// ---- GVLs/kitting deca/axis/AxisHMI_Ex.TcVIS
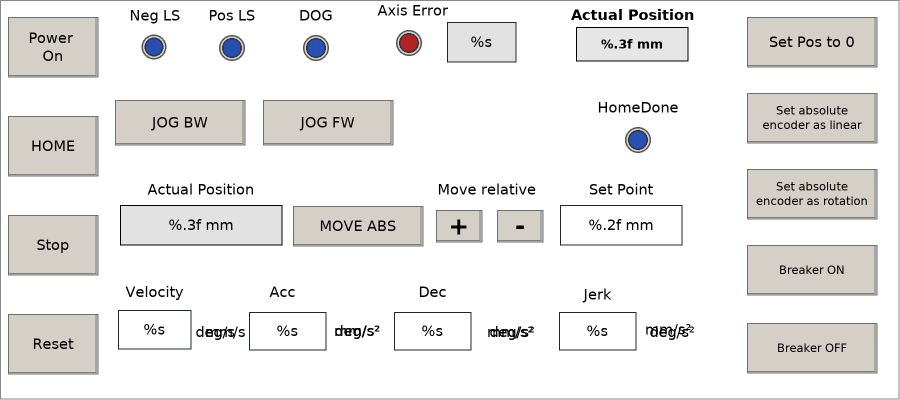
VISUALIZATION AxisHMI_Ex  // 900x400
VAR_IN_OUT
	stAxisHMI	: ST_MotionAxis_MC	;
	mcAxis		: FB_MotionAxis_MC;
	//sAxisName	: STRING			;// Axis Name
	//iAxisID		: INT			;// Axis Id
	xError		: BOOL				;// Axis error flag
END_VAR
    Button (115,100 130x45), "JOG BW", colour toggle: stAxisHMI.mcJog.JogBackwards
        OnMouseDown: execute { stAxisHMI.mcJog.JogBackwards := TRUE; }
        OnMouseUp: execute { stAxisHMI.mcJog.JogBackwards := FALSE; }
    Button (263,100 130x45), "JOG FW", colour toggle: stAxisHMI.mcJog.JogForward
        OnMouseDown: execute { stAxisHMI.mcJog.JogForward := TRUE; }
        OnMouseUp: execute { stAxisHMI.mcJog.JogForward := FALSE; }
    Rectangle (120,205 162x40), "%.3f mm", text variable: stAxisHMI.rActualPosHMI
        OnMouseClick: write the text variable via Default
    Label (141,177 120x25), "Actual Position"
    Button (8,17 90x60), "Power On", colour toggle: stAxisHMI.mcPower.Enable, pressed state: stAxisHMI.mcPower.Enable
        OnMouseClick: toggle stAxisHMI.mcPower.Enable
    Button (8,215 90x60), "Stop", colour toggle: stAxisHMI.mcStop.Execute, invisible if: NOT stAxisHMI.bStopButtonShow
        OnMouseDown: execute { stAxisHMI.mcStop.Execute := TRUE; }
        OnMouseUp: execute { stAxisHMI.mcStop.Execute := FALSE; }
    Button (8,314 90x60), "Reset", colour toggle: stAxisHMI.mcReset.Execute
        OnMouseDown: execute { stAxisHMI.mcReset.Execute := TRUE; }
        OnMouseUp: execute { stAxisHMI.mcReset.Execute := FALSE; }
    Label (111,277 87x30), "Velocity"
    Rectangle (118,310 73x39), "%s", text variable: stAxisHMI.rVeloPers
        OnMouseClick: write the text variable via Default, min 1, max stAxisHMI.rMaxVelocity
    Label (230,277 105x30), "Acc"
    Rectangle (249,312 77x38), "%s", text variable: stAxisHMI.rAcceleration
        OnMouseClick: write stAxisHMI.rAccPers via Default, min 1, max stAxisHMI.rMaxAcceleration
    Lamp1 (139,33 30x28), variable: stAxisHMI.bNegSen, invisible if: NOT stAxisHMI.bNegSensorShow, style: Lamp-Lamp1-Blue
    Label (364,-2 102x25), "Axis Error"
    Rectangle (447,22 69x40), "%s", text variable: stAxisHMI.mcReadStatus.ErrorID
    Lamp1 (394,28 30x30), variable: xError, style: Lamp-Lamp1-Red
    Lamp1 (217,33 30x30), variable: stAxisHMI.bPosSen, invisible if: NOT stAxisHMI.bPosSensorShow, style: Lamp-Lamp1-Blue
    Label (188,3 88x25), "Pos LS", invisible if: NOT stAxisHMI.bPosSensorShow
    Label (111,3 88x25), "Neg LS", invisible if: NOT stAxisHMI.bNegSensorShow
    Rectangle (560,205 122x40), "%.2f mm", text variable: stAxisHMI.rDistance
        OnMouseClick: write the text variable via Default, min 0, max stAxisHMI.rMaxDistance
    Button (293,206 130x40), "MOVE ABS", colour toggle: stAxisHMI.mcMoveAbsolute.Busy, pressed state: stAxisHMI.mcMoveAbsolute.Busy
        OnMouseDown: execute { stAxisHMI.bMoveAbsHMI := TRUE; }
        OnMouseUp: execute { stAxisHMI.bMoveAbsHMI := FALSE; }
    Label (561,177 120x25), "Set Point"
    Button (436,210 46x32), "+", colour toggle: stAxisHMI.mcMoveRelative.Busy, pressed state: stAxisHMI.mcMoveRelative.Busy
        OnMouseDown: execute { stAxisHMI.rPosition := stAxisHMI.rDistance; stAxisHMI.mcMoveRelative.Execute := TRUE; }
        OnMouseUp: execute { stAxisHMI.mcMoveRelative.Execute := FALSE; }
    Button (497,210 46x32), "-", colour toggle: stAxisHMI.mcMoveRelative.Busy, pressed state: stAxisHMI.mcMoveRelative.Busy
        OnMouseDown: execute { stAxisHMI.rPosition := -(stAxisHMI.rDistance); stAxisHMI.mcMoveRelative.Execute := TRUE; }
        OnMouseUp: execute { stAxisHMI.mcMoveRelative.Execute := FALSE; }
    Label (427,177 120x25), "Move relative"
    Label (330,316 55x30), "mm/s²"
    Label (196,317 59x30), "mm/s"
    Label (191,317 49x30), "deg/s", invisible if: NOT stAxisHMI.bUnitDegShow
    Label (328,316 59x30), "deg/s²", invisible if: NOT stAxisHMI.bUnitDegShow
    Label (380,277 105x30), "Dec"
    Rectangle (394,312 77x38), "%s", text variable: stAxisHMI.rDeceleration
        OnMouseClick: write stAxisHMI.rDecPers via Default, min 1, max stAxisHMI.rMaxDeceleration
    Label (483,317 55x30), "mm/s²"
    Label (483,317 59x30), "deg/s²", invisible if: NOT stAxisHMI.bUnitDegShow
    Button (8,116 90x60), "HOME", colour toggle: stAxisHMI.mcHome.Busy
        OnMouseDown: execute { mcAxis.mcHomeAxis.xExecute	:= TRUE; }
        OnMouseUp: execute { mcAxis.mcHomeAxis.xExecute	:= FALSE; }
    Rectangle (559,312 77x38), "%s", text variable: stAxisHMI.rJerk, invisible if: NOT stAxisHMI.bJerkShow
        OnMouseClick: write the text variable via Default, min 0, max stAxisHMI.rMaxJerk
    Label (572,282 51x25), "Jerk", invisible if: NOT stAxisHMI.bJerkShow
    Label (643,317 59x30), "deg/s²", invisible if: NOT stAxisHMI.bUnitDegShow
    Label (641,317 55x25), "mm/s²", invisible if: NOT stAxisHMI.bJerkShow
    Label (557,0 152x30), "Actual Position"
    Rectangle (576,27 112x34), "%.3f mm", text variable: stAxisHMI.rActualPos
    Lamp1 (301,33 30x30), variable: stAxisHMI.bPositionSensor, style: Lamp-Lamp1-Blue
    Label (272,3 88x25), "DOG", invisible if: NOT stAxisHMI.bPosSensorShow
    Lamp1 (623,125 30x30), variable: stAxisHMI.xHomingDone, style: Lamp-Lamp1-Blue
    Label (594,95 88x25), "HomeDone", invisible if: NOT stAxisHMI.bPosSensorShow
    Button (747,17 130x50), "Set Pos to 0", colour toggle: stAxisHMI.CoeWrt.bExecute
        OnMouseDown: execute {
            (*stAxisHMI.CoeWrt.bExecute := TRUE;
            stAxisHMI.nIndex	:= 16#2005;
            stAxisHMI.nSubIndex	:= 16#1F;
            stAxisHMI.iSdoWrite	:= 6;//clear encoder and set current position as origin*)
            stAxisHMI.mcPower.Enable	:= FALSE;
        }
        OnMouseUp: execute { stAxisHMI.iCoeWrt	:= 1; }
    Button (747,93 130x50), "Set absolute encoder as linear", colour toggle: stAxisHMI.CoeWrt.bExecute
        OnMouseDown: execute {
            (*stAxisHMI.CoeWrt.bExecute := TRUE;
            stAxisHMI.nIndex	:= 16#2002;
            stAxisHMI.nSubIndex	:= 16#02;
            stAxisHMI.iSdoWrite	:= 1;//linear mode*)
            stAxisHMI.mcPower.Enable	:= FALSE;
        }
        OnMouseUp: execute { (*stAxisHMI.CoeWrt.bExecute := FALSE;*) stAxisHMI.iCoeWrt	:= 2; }
    Button (747,169 130x50), "Set absolute encoder as rotation", colour toggle: stAxisHMI.CoeWrt.bExecute
        OnMouseDown: execute {
            (*stAxisHMI.CoeWrt.bExecute := TRUE;
            stAxisHMI.nIndex	:= 16#2002;
            stAxisHMI.nSubIndex	:= 16#02;
            stAxisHMI.iSdoWrite	:= 2;//rotate mode*)
            stAxisHMI.mcPower.Enable	:= FALSE;
        }
        OnMouseUp: execute { (*stAxisHMI.CoeWrt.bExecute := FALSE;*) stAxisHMI.iCoeWrt	:= 3; }
    Button (747,245 130x50), "Breaker ON", colour toggle: stAxisHMI.CoeWrt.bExecute
        OnMouseDown: execute {
            (*stAxisHMI.CoeWrt.bExecute := TRUE;
            stAxisHMI.nIndex	:= 16#2004;
            stAxisHMI.nSubIndex	:= 16#06;
            stAxisHMI.iSdoWrite	:= 1;//rotate mode*)
        }
        OnMouseUp: execute { (*stAxisHMI.CoeWrt.bExecute := FALSE;*) stAxisHMI.iCoeWrt	:= 4; }
    Button (747,323 130x50), "Breaker OFF", colour toggle: stAxisHMI.CoeWrt.bExecute
        OnMouseDown: execute {
            (*stAxisHMI.CoeWrt.bExecute := TRUE;
            stAxisHMI.nIndex	:= 16#2004;
            stAxisHMI.nSubIndex	:= 16#06;
            stAxisHMI.iSdoWrite	:= 0;//*)
        }
        OnMouseUp: execute { (*stAxisHMI.CoeWrt.bExecute := FALSE;*) stAxisHMI.iCoeWrt	:= 5; }
END_VISUALIZATION

// ---- VISUs/OtherList.TcVIS
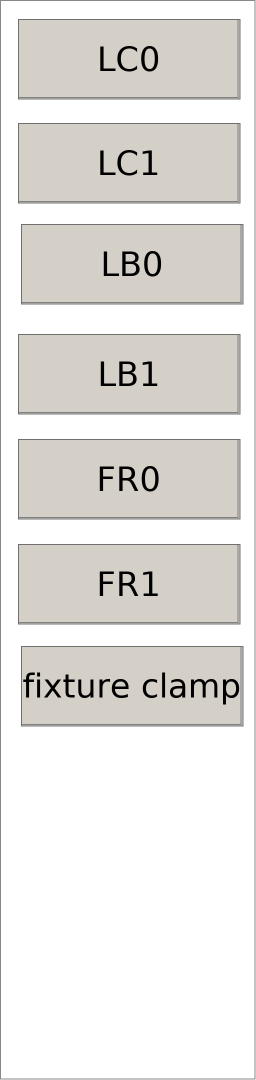
VISUALIZATION OtherList  // 256x1080
    Button (18,19 222x80), "LC0", colour toggle: G_HMI.iOthers =0
        p573394764: 16#FF00FF00
        OnMouseDown: execute {
            G_HMI.iLc  := 0;
            G_HMI.iMainFrame	:= 2;
            G_HMI.iOthers	:= 0;
        }
    Button (21,224 222x80), "LB0", colour toggle: G_HMI.iOthers =2
        p573394764: 16#FF00FF00
        OnMouseDown: execute {
            G_HMI.iLb  := 0;
            G_HMI.iMainFrame	:= 3;
            G_HMI.iOthers	:= 2;
        }
    Button (18,123 222x80), "LC1", colour toggle: G_HMI.iOthers =1
        p573394764: 16#FF00FF00
        OnMouseDown: execute {
            G_HMI.iLc  := 1;
            G_HMI.iMainFrame	:= 2;
            G_HMI.iOthers	:= 1;
        }
    Button (18,334 222x80), "LB1", colour toggle: G_HMI.iOthers =3
        p573394764: 16#FF00FF00
        OnMouseDown: execute {
            G_HMI.iLb  := 1;
            G_HMI.iMainFrame	:= 3;
            G_HMI.iOthers	:= 3;
        }
    Button (18,439 222x80), "FR0", colour toggle: G_HMI.iOthers =4
        p573394764: 16#FF00FF00
        OnMouseDown: execute {
            G_HMI.iFr  := 0;
            G_HMI.iMainFrame	:= 4;
            G_HMI.iOthers	:= 4;
        }
    Button (18,544 222x80), "FR1", colour toggle: G_HMI.iOthers =5
        p573394764: 16#FF00FF00
        OnMouseDown: execute {
            G_HMI.iFr  := 1;
            G_HMI.iMainFrame	:= 4;
            G_HMI.iOthers	:= 5;
        }
    Button (21,646 222x80), "fixture clamp", colour toggle: G_HMI.iOthers =6
        p573394764: 16#FF00FF00
        OnMouseDown: execute { G_HMI.iMainFrame	:= 5; G_HMI.iOthers	:= 6; }
END_VISUALIZATION

// ---- VISUs/visu_LC.TcVIS
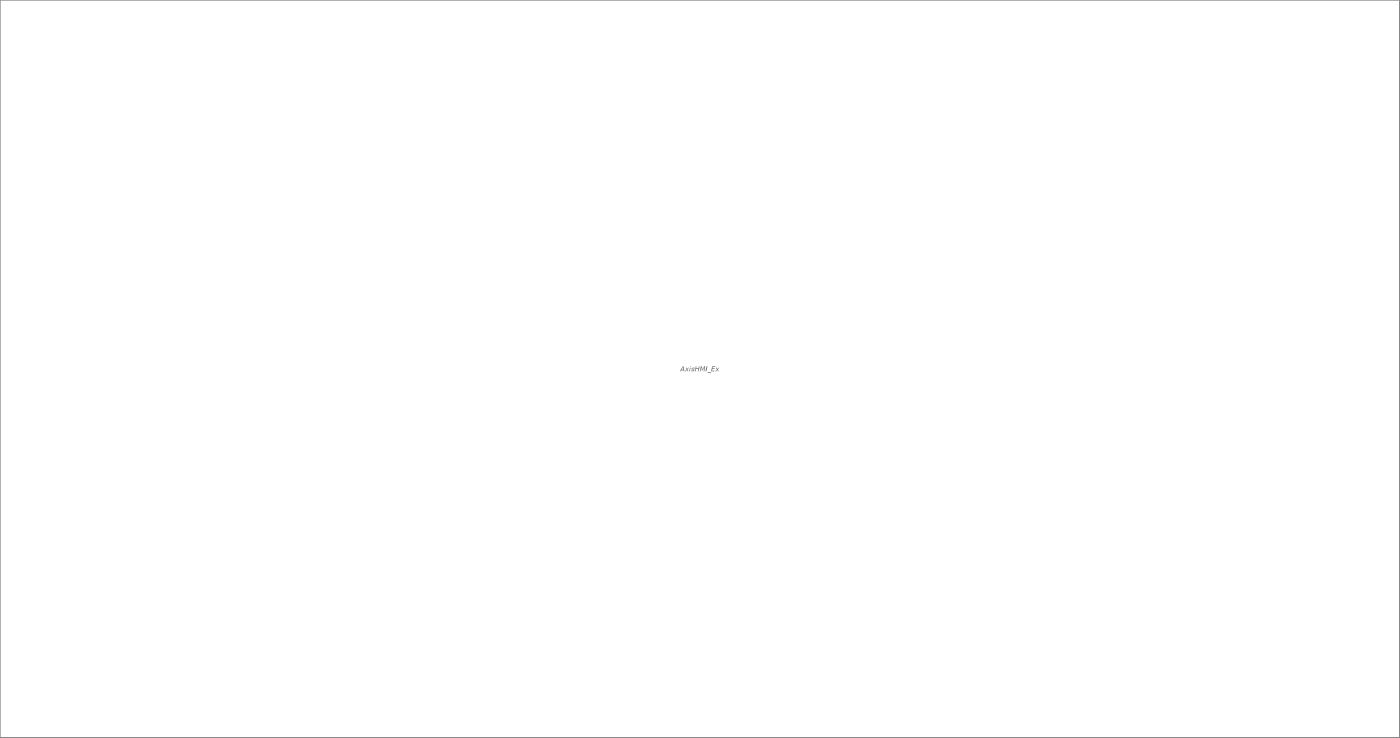
VISUALIZATION visu_LC  // 2048x1080
    TabControl (0,0 2048x1080)
        shows AxisHMI_Ex(stAxisHMI := GVL.lc[G_HMI.iLc].lateral.st_mcAxis, mcAxis := GVL.lc[G_HMI.iLc].lateral.mcAxis, xError := GVL.lc[G_HMI.iLc].lateral.mcAxis.xError)
        shows v_IO_LC(dIO_LC := GVL.lc[G_HMI.iLc])
        shows Axis_HMI(st_axis_HMI := st_mcAxis[EN_Axis.Grip_axis])
        shows v_IO_LC()
        shows v_lc(dIO_LC := GVL.lc[1])
        [0]: TabTitle=LC_axis
        [6]: TabTitle=Gripper
        [1]: AxisHMI=gantrybase.st_mcAxis[EN_Axis.Y], mcAxis=gantrybase.mcAxis[EN_Axis.Y], Error=gantrybase.mcAxis[EN_Axis.Y].xError
        [2]: AxisHMI=gantrybase.st_mcAxis[EN_Axis.Z], mcAxis=gantrybase.mcAxis[EN_Axis.Z], Error=gantrybase.mcAxis[EN_Axis.Z].xError
        p699000190: gantrybase.st_mcAxis[EN_Axis.X]
        p2837713833: gantrybase.mcAxis[EN_Axis.Z].sAxisName
        p520277221: gantrybase.mcAxis[EN_Axis.X].xError
        p3331604638: gantrybase.st_mcAxis[EN_Axis.Z]
        p1813558639: gantrybase.mcAxis[EN_Axis.Z].xError
        p1563495665: gantrybase.st_mcAxis[EN_Axis.Y]
        p2070126892: gantrybase.mcAxis[EN_Axis.Y].xError
        p3435970784: gantrybase.mcAxis[EN_Axis.X]
        p2829954345: gantrybase.mcAxis[EN_Axis.Y]
        p3218520426: gantrybase.mcAxis[EN_Axis.Z]
        p4285860315: GVL.rem[G_HMI.iReM]
        p1681814995: GVL.lc[0]
END_VISUALIZATION

// ---- VISUs/visu_FR.TcVIS
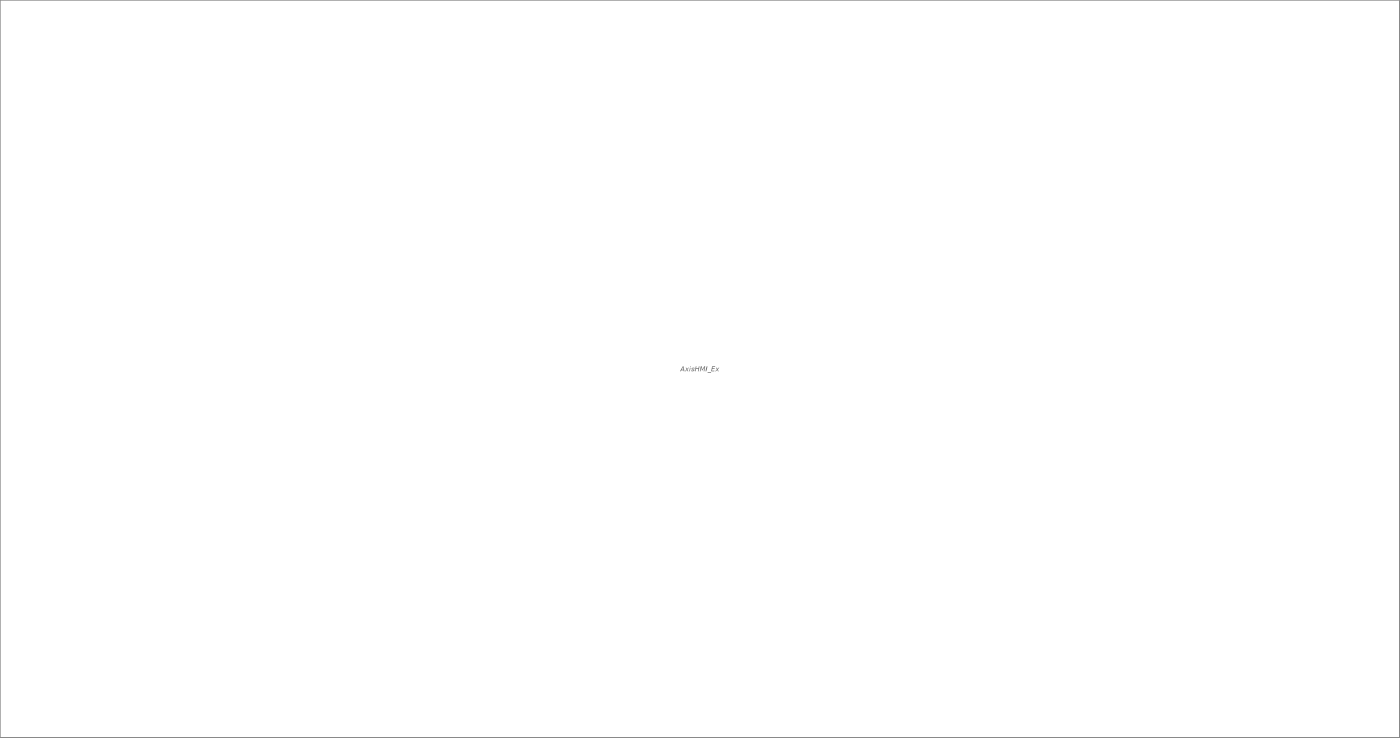
VISUALIZATION visu_FR  // 2048x1080
    TabControl (0,0 2048x1080)
        shows AxisHMI_Ex(stAxisHMI := GVL.fr[G_HMI.iFr].st_mcAxis, mcAxis := GVL.fr[G_HMI.iFr].mcAxis, xError := GVL.fr[G_HMI.iFr].mcAxis.xError)
        shows v_IO_FR(dIO_FR := GVL.fr[G_HMI.iFr])
        shows Axis_HMI(st_axis_HMI := st_mcAxis[EN_Axis.Grip_axis])
        shows v_IO_LC()
        shows v_lc(dIO_LC := GVL.lc[1])
        [0]: TabTitle=FR_axis
        [6]: TabTitle=Gripper
        [1]: AxisHMI=gantrybase.st_mcAxis[EN_Axis.Y], mcAxis=gantrybase.mcAxis[EN_Axis.Y], Error=gantrybase.mcAxis[EN_Axis.Y].xError
        [2]: AxisHMI=gantrybase.st_mcAxis[EN_Axis.Z], mcAxis=gantrybase.mcAxis[EN_Axis.Z], Error=gantrybase.mcAxis[EN_Axis.Z].xError
        p699000190: gantrybase.st_mcAxis[EN_Axis.X]
        p2837713833: gantrybase.mcAxis[EN_Axis.Z].sAxisName
        p520277221: gantrybase.mcAxis[EN_Axis.X].xError
        p3331604638: gantrybase.st_mcAxis[EN_Axis.Z]
        p1813558639: gantrybase.mcAxis[EN_Axis.Z].xError
        p1563495665: gantrybase.st_mcAxis[EN_Axis.Y]
        p2070126892: gantrybase.mcAxis[EN_Axis.Y].xError
        p3435970784: gantrybase.mcAxis[EN_Axis.X]
        p2829954345: gantrybase.mcAxis[EN_Axis.Y]
        p3218520426: gantrybase.mcAxis[EN_Axis.Z]
        p4285860315: GVL.rem[G_HMI.iReM]
        p1681814995: GVL.lc[0]
END_VISUALIZATION

// ---- VISUs/visu_LB.TcVIS
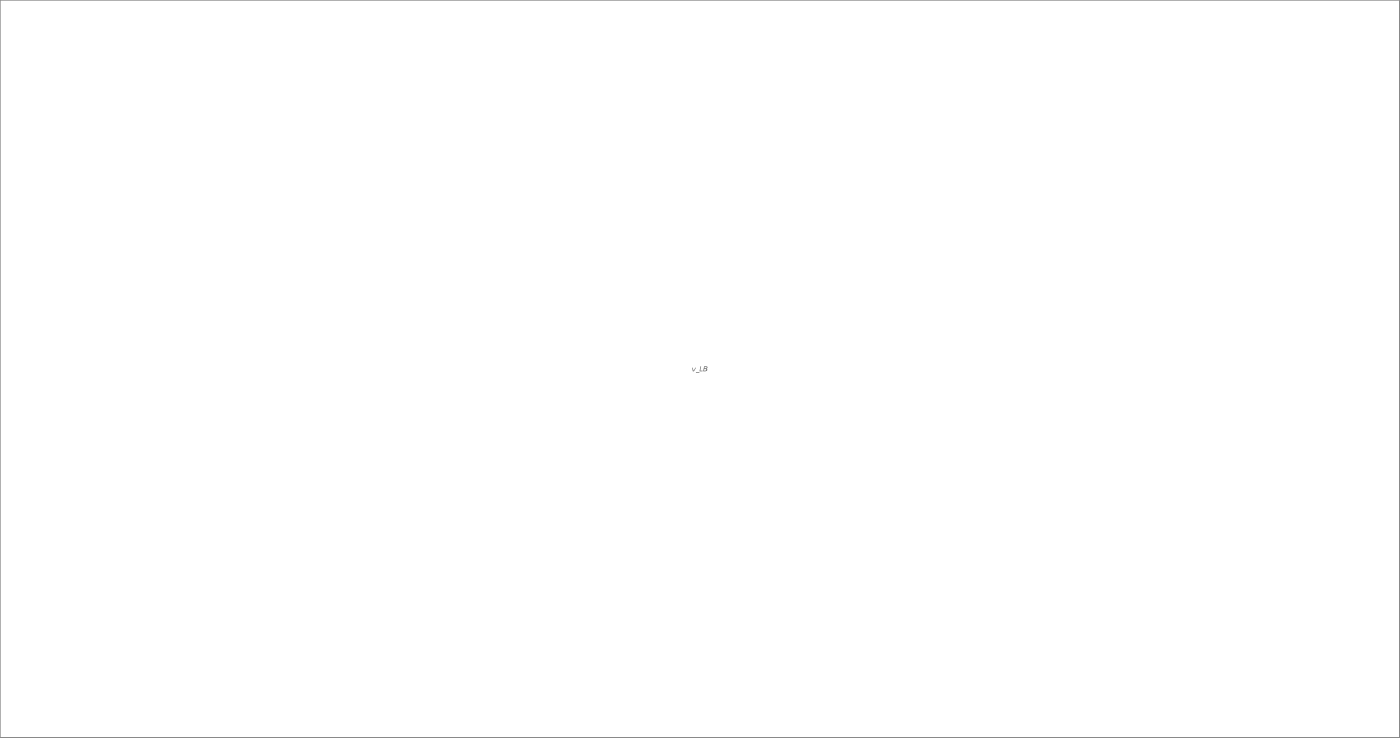
VISUALIZATION visu_LB  // 2048x1080
    TabControl (0,0 2048x1080)
        shows v_LB(dIO_LB := GVL.lb[G_HMI.iLb])
        shows Axis_HMI(st_axis_HMI := st_mcAxis[EN_Axis.Grip_axis])
        shows v_IO_LC(dIO_LC := GVL.lc[G_HMI.iLc])
        shows v_IO_LC()
        shows v_lc(dIO_LC := GVL.lc[1])
        [6]: TabTitle=Gripper
        [1]: AxisHMI=gantrybase.st_mcAxis[EN_Axis.Y], mcAxis=gantrybase.mcAxis[EN_Axis.Y], Error=gantrybase.mcAxis[EN_Axis.Y].xError
        [2]: AxisHMI=gantrybase.st_mcAxis[EN_Axis.Z], mcAxis=gantrybase.mcAxis[EN_Axis.Z], Error=gantrybase.mcAxis[EN_Axis.Z].xError
        p699000190: gantrybase.st_mcAxis[EN_Axis.X]
        p2837713833: gantrybase.mcAxis[EN_Axis.Z].sAxisName
        p520277221: gantrybase.mcAxis[EN_Axis.X].xError
        p3331604638: gantrybase.st_mcAxis[EN_Axis.Z]
        p1813558639: gantrybase.mcAxis[EN_Axis.Z].xError
        p1563495665: gantrybase.st_mcAxis[EN_Axis.Y]
        p2070126892: gantrybase.mcAxis[EN_Axis.Y].xError
        p3435970784: gantrybase.mcAxis[EN_Axis.X]
        p2829954345: gantrybase.mcAxis[EN_Axis.Y]
        p3218520426: gantrybase.mcAxis[EN_Axis.Z]
        p4285860315: GVL.rem[G_HMI.iReM]
        p1681814995: GVL.lc[0]
END_VISUALIZATION

// ---- VISUs/visu_Others.TcVIS
VISUALIZATION visu_Others  // 2048x1080
END_VISUALIZATION

// ---- VISUs/visu_ReM.TcVIS
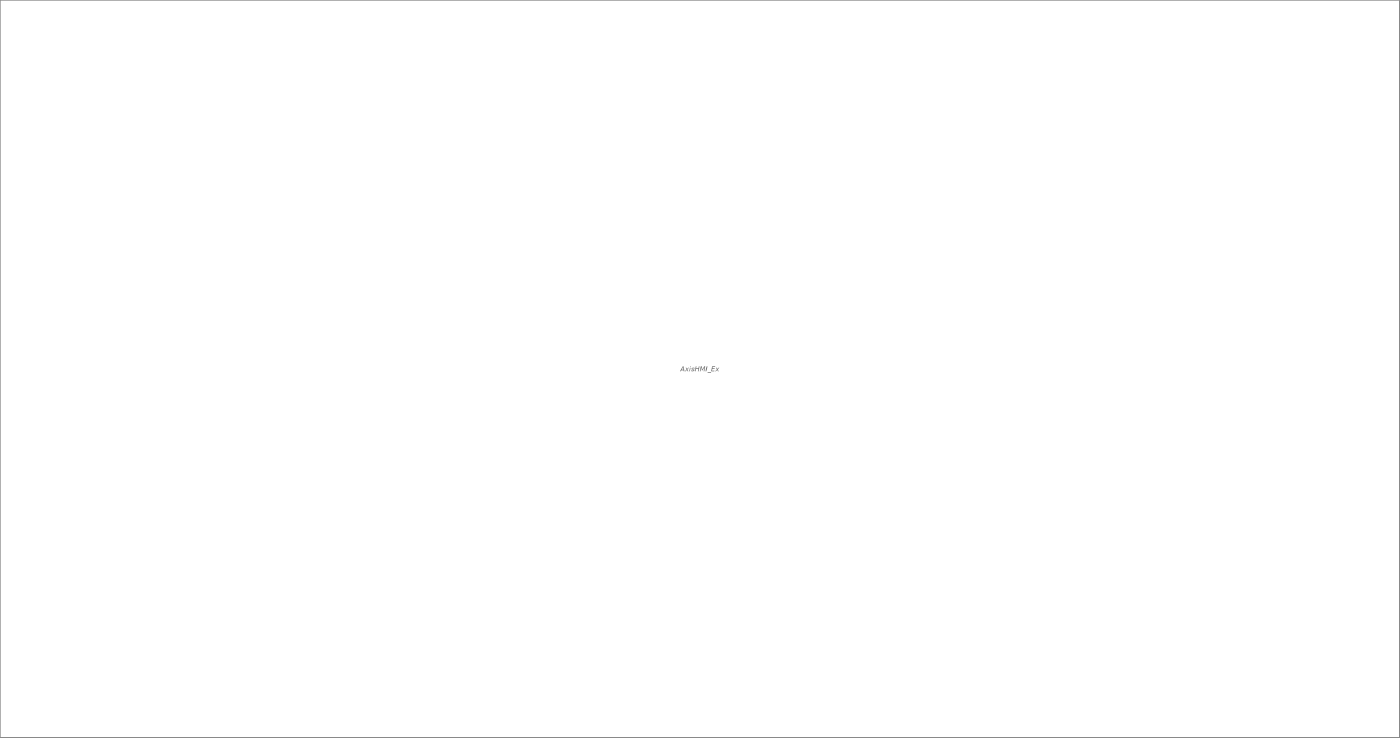
VISUALIZATION visu_ReM  // 2048x1080
    TabControl (0,0 2048x1080)
        shows AxisHMI_Ex(stAxisHMI := GVL.rem[G_HMI.iReM].lift[0].st_mcAxis, mcAxis := GVL.rem[G_HMI.iReM].lift[0].mcAxis, xError := GVL.rem[G_HMI.iReM].lift[0].mcAxis.xError)
        shows AxisHMI_Ex(stAxisHMI := GVL.rem[G_HMI.iReM].lift[1].st_mcAxis, mcAxis := GVL.rem[G_HMI.iReM].lift[1].mcAxis, xError := GVL.rem[G_HMI.iReM].lift[1].mcAxis.xError)
        shows v_rem_0(dIO_ReM := GVL.rem[G_HMI.iReM])
        shows v_rem_1(dIO_ReM := GVL.rem[G_HMI.iReM])
        shows Axis_HMI(st_axis_HMI := st_mcAxis[EN_Axis.Grip_axis])
        [0]: TabTitle=Lift0
        [1]: TabTitle=Lift1
        [2]: TabTitle=ReMIO_0, AxisHMI=gantrybase.st_mcAxis[EN_Axis.Z], mcAxis=gantrybase.mcAxis[EN_Axis.Z], Error=gantrybase.mcAxis[EN_Axis.Z].xError
        [3]: TabTitle=ReMIO_1
        [6]: TabTitle=Gripper
        p699000190: gantrybase.st_mcAxis[EN_Axis.X]
        p2837713833: gantrybase.mcAxis[EN_Axis.Z].sAxisName
        p520277221: gantrybase.mcAxis[EN_Axis.X].xError
        p3331604638: gantrybase.st_mcAxis[EN_Axis.Z]
        p1813558639: gantrybase.mcAxis[EN_Axis.Z].xError
        p1563495665: gantrybase.st_mcAxis[EN_Axis.Y]
        p2070126892: gantrybase.mcAxis[EN_Axis.Y].xError
        p3435970784: gantrybase.mcAxis[EN_Axis.X]
        p2829954345: gantrybase.mcAxis[EN_Axis.Y]
        p3218520426: gantrybase.mcAxis[EN_Axis.Z]
END_VISUALIZATION

// ---- VISUs/visu_MLC.TcVIS
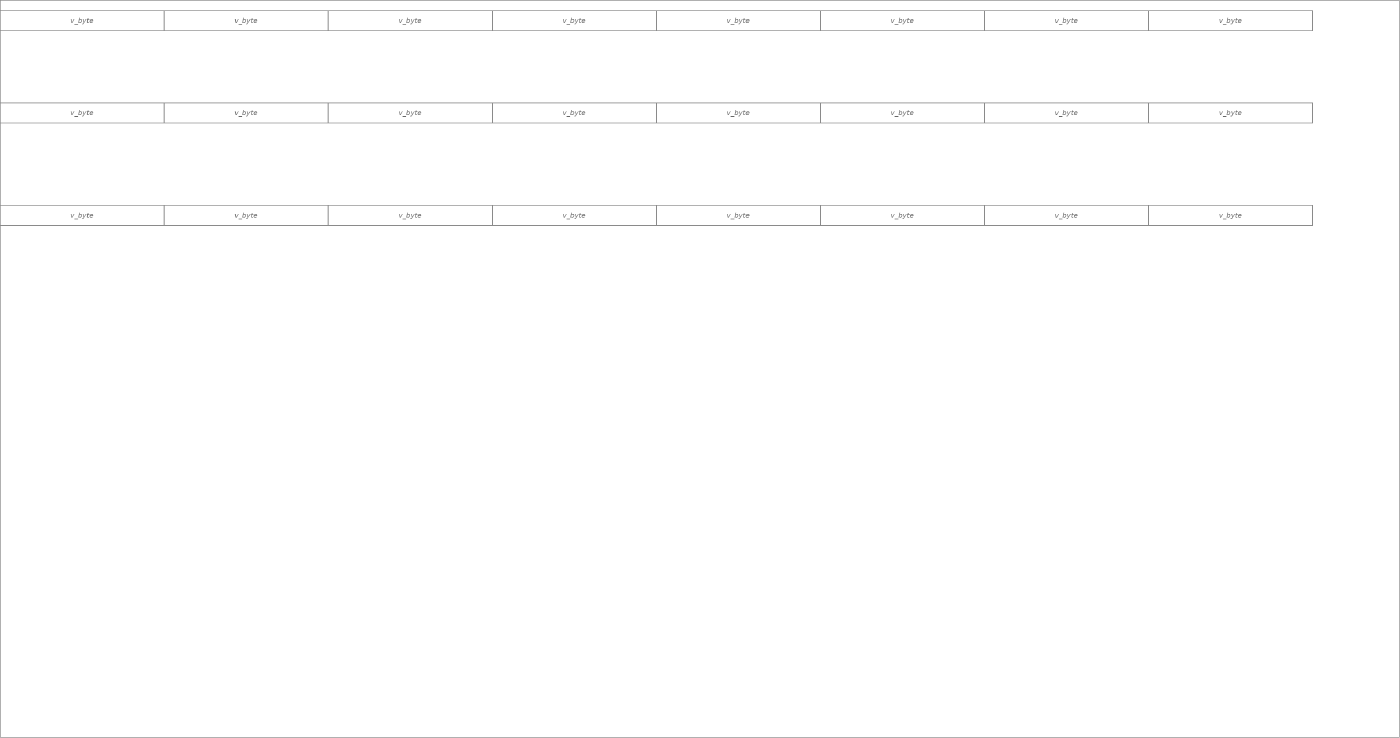
VISUALIZATION visu_MLC  // 2048x1080
    Frame (0,15 240x30)
        shows v_byte(iNum := GVL.ibyteNum[1])
    Frame (0,300 240x30)
        shows v_byte(iNum := GVL.ibyteNum[17])
    Frame (240,300 240x30)
        shows v_byte(iNum := GVL.ibyteNum[18])
    Frame (480,300 240x30)
        shows v_byte(iNum := GVL.ibyteNum[19])
    Frame (720,300 240x30)
        shows v_byte(iNum := GVL.ibyteNum[20])
    Frame (960,300 240x30)
        shows v_byte(iNum := GVL.ibyteNum[21])
    Frame (1200,300 240x30)
        shows v_byte(iNum := GVL.ibyteNum[22])
    Frame (1440,300 240x30)
        shows v_byte(iNum := GVL.ibyteNum[23])
    Frame (1680,300 240x30)
        shows v_byte(iNum := GVL.ibyteNum[24])
    Frame (0,150 240x30)
        shows v_byte(iNum := GVL.ibyteNum[9])
    Frame (240,150 240x30)
        shows v_byte(iNum := GVL.ibyteNum[10])
    Frame (480,150 240x30)
        shows v_byte(iNum := GVL.ibyteNum[11])
    Frame (720,150 240x30)
        shows v_byte(iNum := GVL.ibyteNum[12])
    Frame (960,150 240x30)
        shows v_byte(iNum := GVL.ibyteNum[13])
    Frame (1200,150 240x30)
        shows v_byte(iNum := GVL.ibyteNum[14])
    Frame (1440,150 240x30)
        shows v_byte(iNum := GVL.ibyteNum[15])
    Frame (1680,150 240x30)
        shows v_byte(iNum := GVL.ibyteNum[16])
    Frame (240,15 240x30)
        shows v_byte(iNum := GVL.ibyteNum[2])
    Frame (480,15 240x30)
        shows v_byte(iNum := GVL.ibyteNum[3])
    Frame (720,15 240x30)
        shows v_byte(iNum := GVL.ibyteNum[4])
    Frame (960,15 240x30)
        shows v_byte(iNum := GVL.ibyteNum[5])
    Frame (1200,15 240x30)
        shows v_byte(iNum := GVL.ibyteNum[6])
    Frame (1440,15 240x30)
        shows v_byte(iNum := GVL.ibyteNum[7])
    Frame (1680,15 240x30)
        shows v_byte(iNum := GVL.ibyteNum[8])
END_VISUALIZATION

// ---- VISUs/visu_main.TcVIS
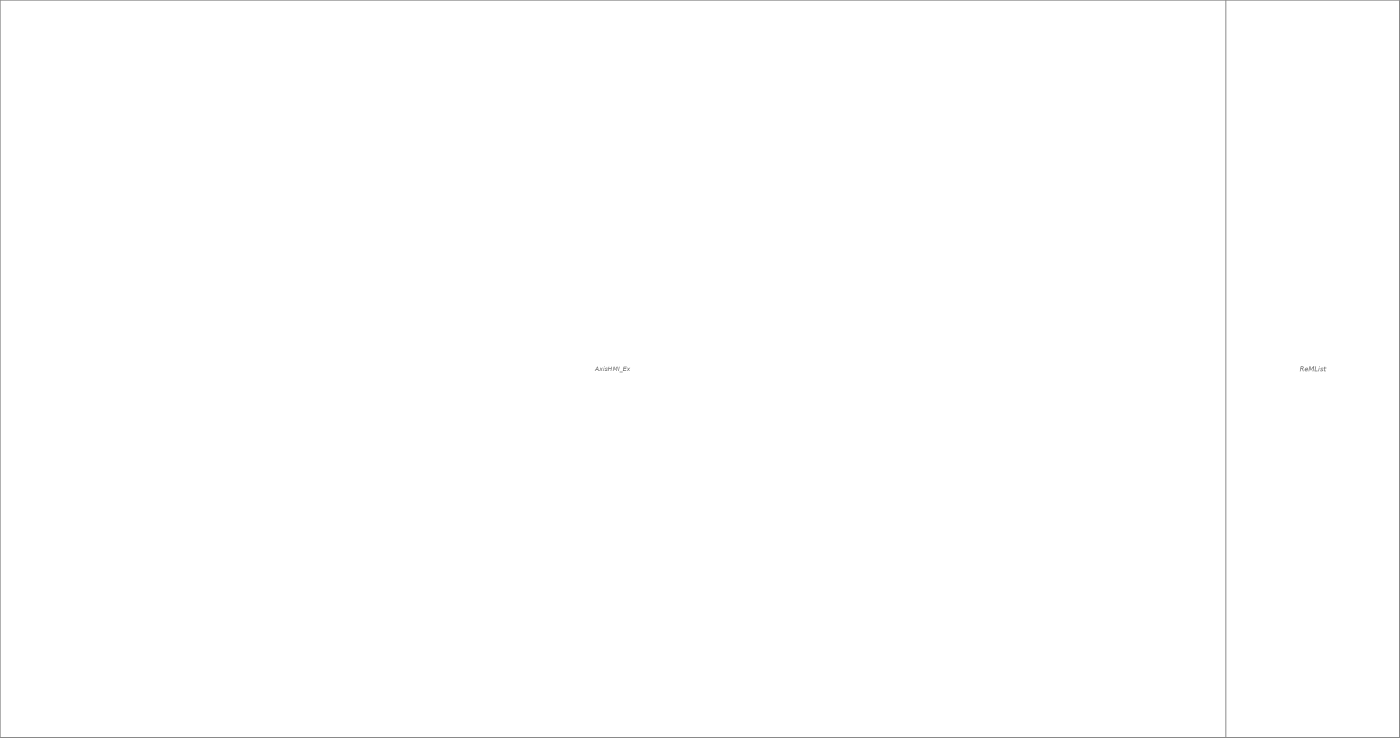
VISUALIZATION visu_main  // 2048x1080
    TabControl (1793,0 255x1080), frame switch variable: G_HMI.iMainFrame
        shows ReMList()
        shows PMList()
        shows OtherList()
        shows Visualization_4()
        [0]: TabTitle=ReM
        [2]: TabTitle=Others
    Frame (0,0 1793x1080), frame switch variable: G_HMI.iMainFrame
        shows visu_ReM()
        shows visu_PM()
        shows visu_LC()
        shows visu_LB()
        shows visu_FR()
        shows v_IO_fixtureClamp()
END_VISUALIZATION

// ---- VISUs/PMList.TcVIS
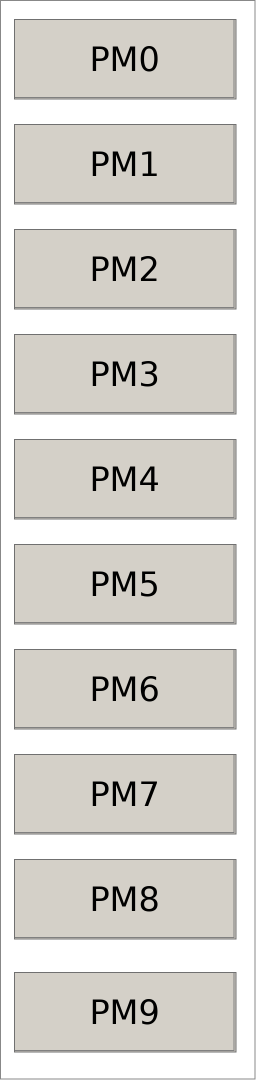
VISUALIZATION PMList  // 256x1080
    Button (14,19 222x80), "PM0", colour toggle: G_HMI.iPM =0
        p573394764: 16#FF00FF00
        OnMouseDown: execute { G_HMI.iPM  := 0; G_HMI.iMainFrame	:= 1; }
    Button (14,124 222x80), "PM1", colour toggle: G_HMI.iPM =1
        p573394764: 16#FF00FF00
        OnMouseDown: execute { G_HMI.iPM  := 1; G_HMI.iMainFrame	:= 1; }
    Button (14,229 222x80), "PM2", colour toggle: G_HMI.iPM =2
        p573394764: 16#FF00FF00
        OnMouseDown: execute { G_HMI.iPM  := 2; G_HMI.iMainFrame	:= 1; }
    Button (14,334 222x80), "PM3", colour toggle: G_HMI.iPM =3
        p573394764: 16#FF00FF00
        OnMouseDown: execute { G_HMI.iPM  := 3; G_HMI.iMainFrame	:= 1; }
    Button (14,439 222x80), "PM4", colour toggle: G_HMI.iPM =4
        p573394764: 16#FF00FF00
        OnMouseDown: execute { G_HMI.iPM  := 4; G_HMI.iMainFrame	:= 1; }
    Button (14,544 222x80), "PM5", colour toggle: G_HMI.iPM =5
        p573394764: 16#FF00FF00
        OnMouseDown: execute { G_HMI.iPM  := 5; G_HMI.iMainFrame	:= 1; }
    Button (14,649 222x80), "PM6", colour toggle: G_HMI.iPM =6
        p573394764: 16#FF00FF00
        OnMouseDown: execute { G_HMI.iPM  := 6; G_HMI.iMainFrame	:= 1; }
    Button (14,754 222x80), "PM7", colour toggle: G_HMI.iPM =7
        p573394764: 16#FF00FF00
        OnMouseDown: execute { G_HMI.iPM  := 7; G_HMI.iMainFrame	:= 1; }
    Button (14,859 222x80), "PM8", colour toggle: G_HMI.iPM =8
        p573394764: 16#FF00FF00
        OnMouseDown: execute { G_HMI.iPM  := 8; G_HMI.iMainFrame	:= 1; }
    Button (14,972 222x80), "PM9", colour toggle: G_HMI.iPM =9
        p573394764: 16#FF00FF00
        OnMouseDown: execute { G_HMI.iPM  := 9; G_HMI.iMainFrame	:= 1; }
END_VISUALIZATION

// ---- VISUs/v_IO_FR.TcVIS
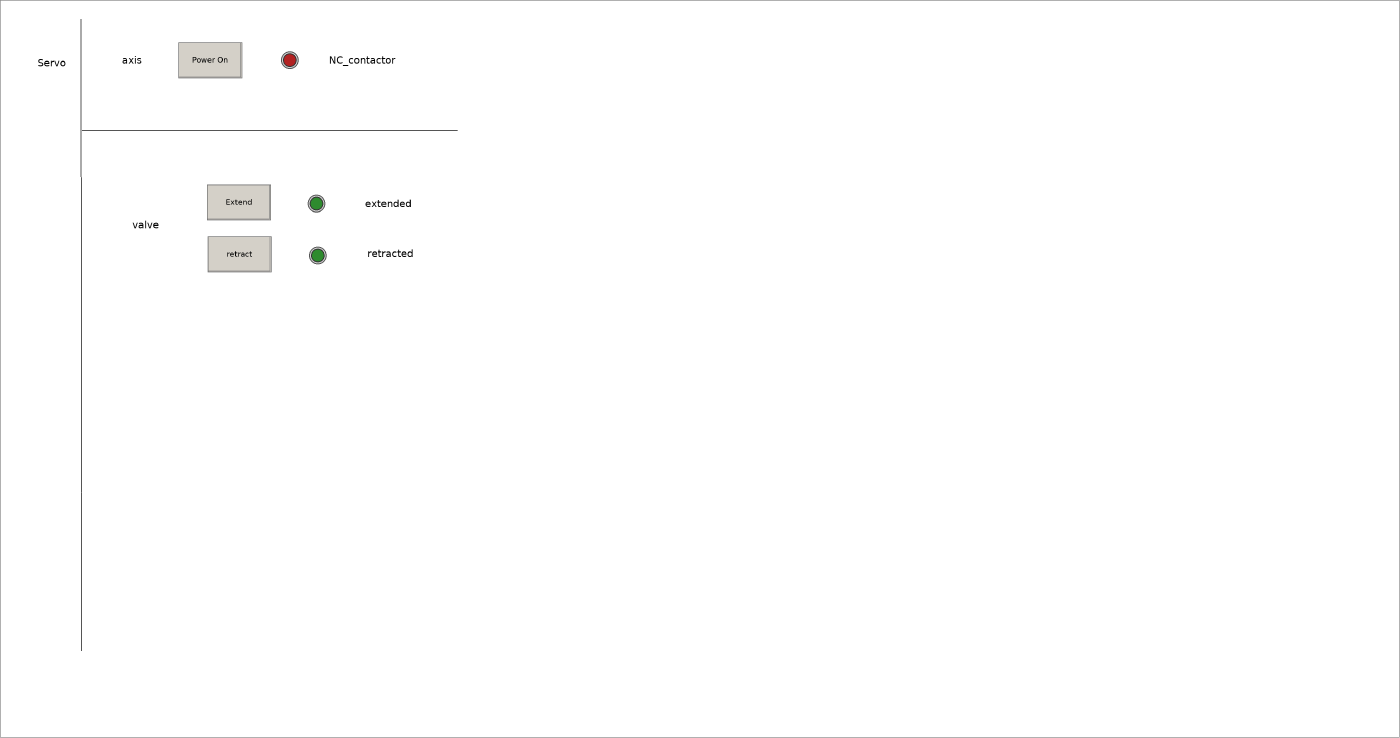
VISUALIZATION v_IO_FR  // 2048x1080
VAR_IN_OUT
	dIO_FR		: fixtureRotation_Module;
END_VAR
    Line (120,190) (669,190)
    Line (118,28) (119,952)
    Label (464,75 132x26), "NC_contactor"
    Label (127,75 132x26), "axis"
    Button (261,62 93x52), "Power On", colour toggle: dIO_FR.power_axis
        toggle dIO_FR.power_axis
    Lamp1 (409,73 30x30), variable: dIO_FR.contactor_axis, style: Lamp-Lamp1-Red
    Label (133,316 160x26), "valve"
    Button (303,270 93x52), "Extend", colour toggle: dIO_FR.valve.extend
        OnMouseDown: execute { dIO_FR.valve.extend := TRUE; dIO_FR.valve.retract := FALSE; }
    Button (304,346 93x52), "retract", colour toggle: dIO_FR.valve.retract
        OnMouseDown: execute { dIO_FR.valve.extend := FALSE; dIO_FR.valve.retract := TRUE; }
    Lamp1 (448,283 30x30), variable: dIO_FR.valve.extended, style: Lamp-Lamp1-Green
    Lamp1 (450,359 30x30), variable: dIO_FR.valve.retracted, style: Lamp-Lamp1-Green
    Label (502,285 132x26), "extended"
    Label (505,358 132x26), "retracted"
    Label (36,79 80x26), "Servo"
END_VISUALIZATION

// ---- VISUs/v_IO_fixtureClamp.TcVIS
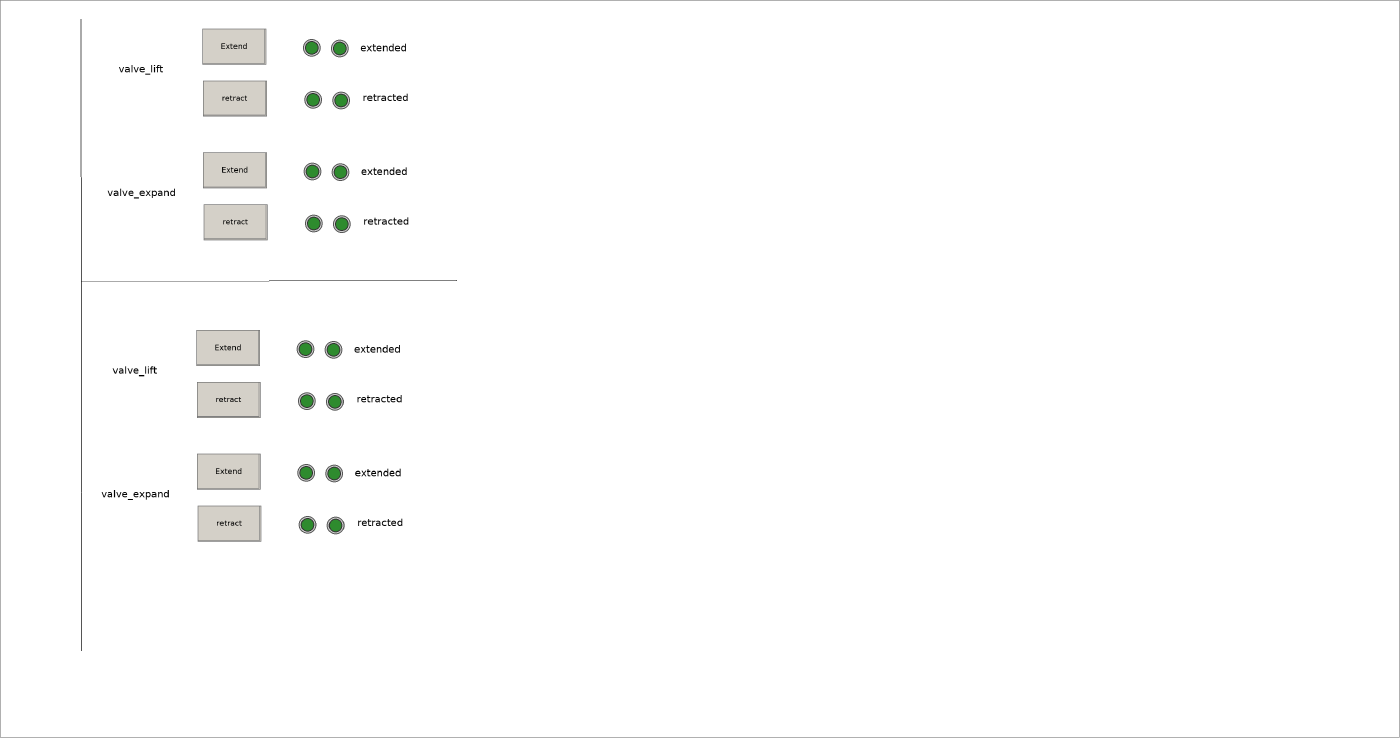
VISUALIZATION v_IO_fixtureClamp  // 2048x1080
    Line (118,28) (119,952)
    Label (126,88 160x26), "valve_lift"
    Button (296,42 93x52), "Extend", colour toggle: G_IO.arDO[55].Ch[10]
        OnMouseDown: execute { G_IO.arDO[55].Ch[10] := TRUE; G_IO.arDO[55].Ch[11] := FALSE; }
    Button (297,118 93x52), "retract", colour toggle: G_IO.arDO[55].Ch[11]
        OnMouseDown: execute { G_IO.arDO[55].Ch[10] := FALSE; G_IO.arDO[55].Ch[11] := TRUE; }
    Lamp1 (441,55 30x30), variable: G_IO.arDI[77].Ch[0], style: Lamp-Lamp1-Green
    Lamp1 (443,131 30x30), variable: G_IO.arDI[77].Ch[1], style: Lamp-Lamp1-Green
    Label (495,57 132x26), "extended"
    Label (498,130 132x26), "retracted"
    Lamp1 (482,56 30x30), variable: G_IO.arDI[77].Ch[2], style: Lamp-Lamp1-Green
    Lamp1 (484,132 30x30), variable: G_IO.arDI[77].Ch[3], style: Lamp-Lamp1-Green
    Label (127,269 160x26), "valve_expand"
    Button (297,223 93x52), "Extend", colour toggle: G_IO.arDO[55].Ch[12]
        OnMouseDown: execute { G_IO.arDO[55].Ch[12] := TRUE; G_IO.arDO[55].Ch[13] := FALSE; }
    Button (298,299 93x52), "retract", colour toggle: G_IO.arDO[55].Ch[13]
        OnMouseDown: execute { G_IO.arDO[55].Ch[12] := FALSE; G_IO.arDO[55].Ch[13] := TRUE; }
    Lamp1 (442,236 30x30), variable: G_IO.arDI[77].Ch[4], style: Lamp-Lamp1-Green
    Lamp1 (444,312 30x30), variable: G_IO.arDI[77].Ch[5], style: Lamp-Lamp1-Green
    Label (496,238 132x26), "extended"
    Label (499,311 132x26), "retracted"
    Lamp1 (483,237 30x30), variable: G_IO.arDI[77].Ch[6], style: Lamp-Lamp1-Green
    Lamp1 (485,313 30x30), variable: G_IO.arDI[77].Ch[7], style: Lamp-Lamp1-Green
    Label (117,529 160x26), "valve_lift"
    Button (287,483 93x52), "Extend", colour toggle: G_IO.arDO[59].Ch[10]
        OnMouseDown: execute { G_IO.arDO[59].Ch[10] := TRUE; G_IO.arDO[59].Ch[11] := FALSE; }
    Button (288,559 93x52), "retract", colour toggle: G_IO.arDO[59].Ch[11]
        OnMouseDown: execute { G_IO.arDO[59].Ch[10] := FALSE; G_IO.arDO[59].Ch[11] := TRUE; }
    Lamp1 (432,496 30x30), variable: G_IO.arDI[78].Ch[0], style: Lamp-Lamp1-Green
    Lamp1 (434,572 30x30), variable: G_IO.arDI[78].Ch[1], style: Lamp-Lamp1-Green
    Label (486,498 132x26), "extended"
    Label (489,571 132x26), "retracted"
    Lamp1 (473,497 30x30), variable: G_IO.arDI[78].Ch[2], style: Lamp-Lamp1-Green
    Lamp1 (475,573 30x30), variable: G_IO.arDI[78].Ch[3], style: Lamp-Lamp1-Green
    Label (118,710 160x26), "valve_expand"
    Button (288,664 93x52), "Extend", colour toggle: G_IO.arDO[59].Ch[12]
        OnMouseDown: execute { G_IO.arDO[59].Ch[12] := TRUE; G_IO.arDO[59].Ch[13] := FALSE; }
    Button (289,740 93x52), "retract", colour toggle: G_IO.arDO[59].Ch[13]
        OnMouseDown: execute { G_IO.arDO[59].Ch[12] := FALSE; G_IO.arDO[59].Ch[13] := TRUE; }
    Lamp1 (433,677 30x30), variable: G_IO.arDI[78].Ch[4], style: Lamp-Lamp1-Green
    Lamp1 (435,753 30x30), variable: G_IO.arDI[78].Ch[5], style: Lamp-Lamp1-Green
    Label (487,679 132x26), "extended"
    Label (490,752 132x26), "retracted"
    Lamp1 (474,678 30x30), variable: G_IO.arDI[78].Ch[6], style: Lamp-Lamp1-Green
    Lamp1 (476,754 30x30), variable: G_IO.arDI[78].Ch[7], style: Lamp-Lamp1-Green
    Line (119,411) (668,410)
END_VISUALIZATION

// ---- VISUs/v_IO_LC.TcVIS
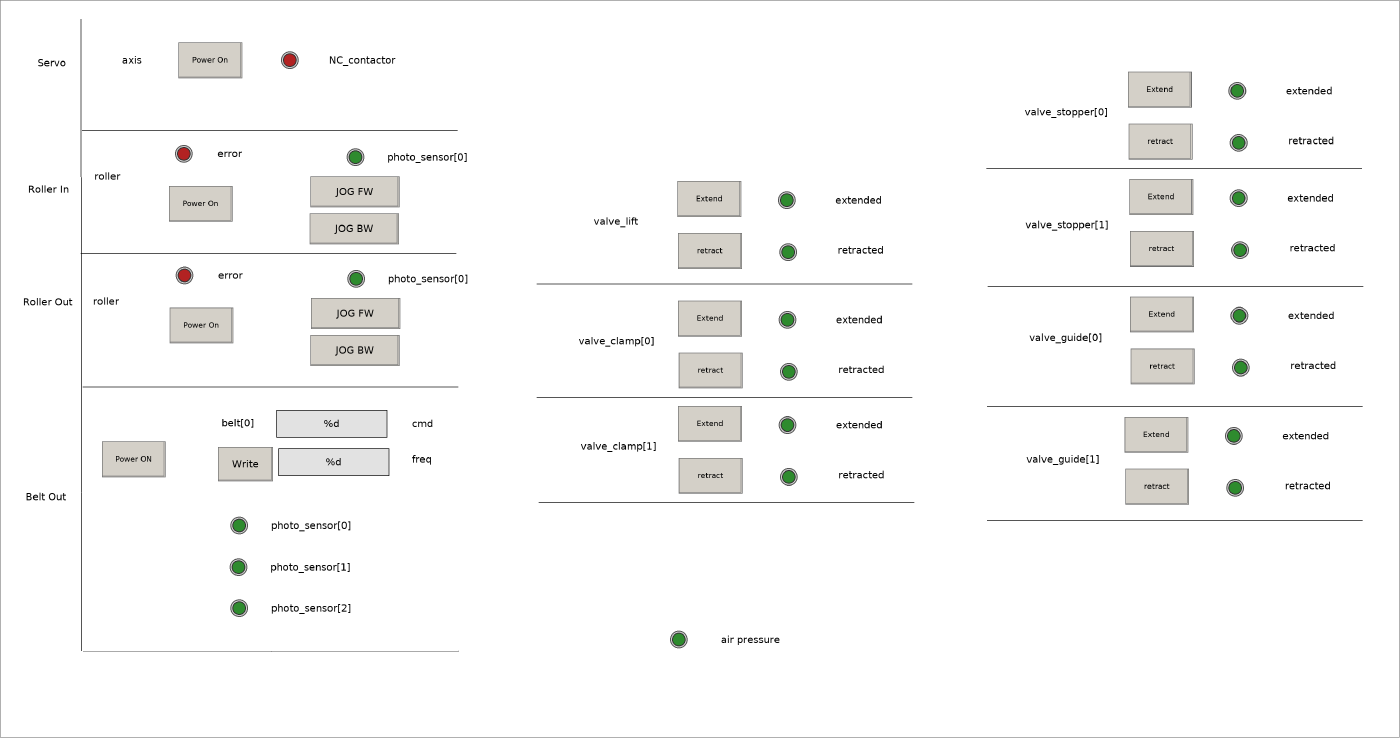
VISUALIZATION v_IO_LC  // 2048x1080
VAR_IN_OUT
	dIO_LC		: LateralRecy_Module;
END_VAR
    Lamp1 (505,215 30x30), variable: dIO_LC.rollerIn.photo_sensor, style: Lamp-Lamp1-Green
    Label (559,217 132x26), "photo_sensor[0]"
    Label (31,264 80x26), "Roller In"
    Lamp1 (254,210 30x30), variable: dIO_LC.rollerIn.roller.err, style: Lamp-Lamp1-Red
    Label (270,212 132x26), "error"
    Label (91,245 132x26), "roller"
    Line (120,190) (669,190)
    Line (118,28) (119,952)
    Button (454,258 130x45), "JOG FW", colour toggle: dIO_LC.rollerIn.roller.forward
        OnMouseDown: execute { dIO_LC.rollerIn.roller.forward := TRUE; }
        OnMouseUp: execute { dIO_LC.rollerIn.roller.forward := FALSE; }
    Button (453,312 130x45), "JOG BW", colour toggle: dIO_LC.rollerIn.roller.backward
        OnMouseDown: execute { dIO_LC.rollerIn.roller.backward := TRUE; }
        OnMouseUp: execute { dIO_LC.rollerIn.roller.backward := FALSE; }
    Button (247,272 93x52), "Power On", colour toggle: dIO_LC.rollerIn.roller.Power
        toggle dIO_LC.rollerIn.roller.Power
    Line (118,370) (667,370)
    Line (121,566) (670,566)
    Label (1480,151 160x26), "valve_stopper[0]"
    Button (1650,105 93x52), "Extend", colour toggle: dIO_LC.valve_stopper[0].extend
        OnMouseDown: execute { dIO_LC.valve_stopper[0].extend := TRUE; dIO_LC.valve_stopper[0].retract := FALSE; }
    Button (1651,181 93x52), "retract", colour toggle: dIO_LC.valve_stopper[0].retract
        OnMouseDown: execute { dIO_LC.valve_stopper[0].extend := FALSE; dIO_LC.valve_stopper[0].retract := TRUE; }
    Lamp1 (1795,118 30x30), variable: dIO_LC.valve_stopper[0].extended, style: Lamp-Lamp1-Green
    Lamp1 (1797,194 30x30), variable: dIO_LC.valve_stopper[0].retracted, style: Lamp-Lamp1-Green
    Label (1849,120 132x26), "extended"
    Label (1852,193 132x26), "retracted"
    Label (1481,316 160x26), "valve_stopper[1]"
    Label (1479,481 160x26), "valve_guide[0]"
    Label (1475,659 160x26), "valve_guide[1]"
    Line (1443,246) (1992,246)
    Line (1445,419) (1994,419)
    Line (1444,594) (1993,594)
    Line (1444,761) (1993,761)
    Label (89,428 132x26), "roller"
    Label (30,429 80x26), "Roller Out"
    Rectangle (404,600 162x40), "%d", text variable: dIO_LC.belt_out.belt.fbconverter.cmd
        OnMouseClick: write the text variable via Default
    Rectangle (407,656 162x40), "%d", text variable: dIO_LC.belt_out.belt.fbconverter.freq
        OnMouseClick: write the text variable via Default
    Label (282,606 132x26), "belt[0]"
    Label (552,607 132x26), "cmd"
    Label (551,659 132x26), "freq"
    Button (149,646 93x52), "Power ON", colour toggle: dIO_LC.power_beltConv
        toggle dIO_LC.power_beltConv
    Button (319,654 80x50), "Write"
        OnMouseDown: execute { dIO_LC.belt_out.belt.fbconverter.bSetParaEx	:= TRUE; }
        OnMouseUp: execute { dIO_LC.belt_out.belt.fbconverter.bSetParaEx	:= FALSE; }
    Lamp1 (335,754 30x30), variable: dIO_LC.belt_out.photo_sensor[0], style: Lamp-Lamp1-Green
    Label (389,756 132x26), "photo_sensor[0]"
    Lamp1 (334,815 30x30), variable: dIO_LC.belt_out.photo_sensor[1], style: Lamp-Lamp1-Green
    Label (388,817 132x26), "photo_sensor[1]"
    Lamp1 (335,875 30x30), variable: dIO_LC.belt_out.photo_sensor[2], style: Lamp-Lamp1-Green
    Label (389,877 132x26), "photo_sensor[2]"
    Label (464,75 132x26), "NC_contactor"
    Label (127,75 132x26), "axis"
    Button (261,62 93x52), "Power On", colour toggle: dIO_LC.lateral.power_axis
        toggle dIO_LC.lateral.power_axis
    Lamp1 (409,73 30x30), variable: dIO_LC.lateral.contactor_axis, style: Lamp-Lamp1-Red
    Label (821,311 160x26), "valve_lift"
    Button (991,265 93x52), "Extend", colour toggle: dIO_LC.lateral.valve_lift.extend
        OnMouseDown: execute { dIO_LC.lateral.valve_lift.extend := TRUE; dIO_LC.lateral.valve_lift.retract := FALSE; }
    Button (992,341 93x52), "retract", colour toggle: dIO_LC.lateral.valve_lift.retract
        OnMouseDown: execute { dIO_LC.lateral.valve_lift.extend := FALSE; dIO_LC.lateral.valve_lift.retract := TRUE; }
    Lamp1 (1136,278 30x30), variable: dIO_LC.lateral.valve_lift.extended, style: Lamp-Lamp1-Green
    Lamp1 (1138,354 30x30), variable: dIO_LC.lateral.valve_lift.retracted, style: Lamp-Lamp1-Green
    Label (1190,280 132x26), "extended"
    Label (1193,353 132x26), "retracted"
    Label (822,486 160x26), "valve_clamp[0]"
    Button (992,440 93x52), "Extend", colour toggle: dIO_LC.lateral.valve_clamp[0].extend
        OnMouseDown: execute { dIO_LC.lateral.valve_clamp[0].extend := TRUE; dIO_LC.lateral.valve_clamp[0].retract := FALSE; }
    Button (993,516 93x52), "retract", colour toggle: dIO_LC.lateral.valve_clamp[0].retract
        OnMouseDown: execute { dIO_LC.lateral.valve_clamp[0].extend := FALSE; dIO_LC.lateral.valve_clamp[0].retract := TRUE; }
    Lamp1 (1137,453 30x30), variable: dIO_LC.lateral.valve_clamp[0].extended, style: Lamp-Lamp1-Green
    Lamp1 (1139,529 30x30), variable: dIO_LC.lateral.valve_clamp[0].retracted, style: Lamp-Lamp1-Green
    Label (1191,455 132x26), "extended"
    Label (1194,528 132x26), "retracted"
    Line (785,581) (1334,581)
    Label (825,640 160x26), "valve_clamp[1]"
    Line (788,735) (1337,735)
    Line (785,415) (1334,415)
    Line (122,953) (671,952)
    Label (27,714 80x26), "Belt Out"
    Label (36,79 80x26), "Servo"
    Lamp1 (506,393 30x30), variable: dIO_LC.rollerOut.photo_sensor, style: Lamp-Lamp1-Green
    Label (560,395 132x26), "photo_sensor[0]"
    Lamp1 (255,388 30x30), variable: dIO_LC.rollerOut.roller.err, style: Lamp-Lamp1-Red
    Label (271,390 132x26), "error"
    Button (455,436 130x45), "JOG FW", colour toggle: dIO_LC.rollerOut.roller.forward
        OnMouseDown: execute { dIO_LC.rollerOut.roller.forward := TRUE; }
        OnMouseUp: execute { dIO_LC.rollerOut.roller.forward := FALSE; }
    Button (454,490 130x45), "JOG BW", colour toggle: dIO_LC.rollerOut.roller.backward
        OnMouseDown: execute { dIO_LC.rollerOut.roller.backward := TRUE; }
        OnMouseUp: execute { dIO_LC.rollerOut.roller.backward := FALSE; }
    Button (248,450 93x52), "Power On", colour toggle: dIO_LC.rollerOut.roller.Power
        toggle dIO_LC.rollerOut.roller.Power
    Button (992,594 93x52), "Extend", colour toggle: dIO_LC.lateral.valve_clamp[1].extend
        OnMouseDown: execute { dIO_LC.lateral.valve_clamp[1].extend := TRUE; dIO_LC.lateral.valve_clamp[1].retract := FALSE; }
    Button (993,670 93x52), "retract", colour toggle: dIO_LC.lateral.valve_clamp[1].retract
        OnMouseDown: execute { dIO_LC.lateral.valve_clamp[1].extend := FALSE; dIO_LC.lateral.valve_clamp[1].retract := TRUE; }
    Lamp1 (1137,607 30x30), variable: dIO_LC.lateral.valve_clamp[1].extended, style: Lamp-Lamp1-Green
    Lamp1 (1139,683 30x30), variable: dIO_LC.lateral.valve_clamp[1].retracted, style: Lamp-Lamp1-Green
    Label (1191,609 132x26), "extended"
    Label (1194,682 132x26), "retracted"
    Button (1652,262 93x52), "Extend", colour toggle: dIO_LC.valve_stopper[1].extend
        OnMouseDown: execute { dIO_LC.valve_stopper[1].extend := TRUE; dIO_LC.valve_stopper[1].retract := FALSE; }
    Button (1653,338 93x52), "retract", colour toggle: dIO_LC.valve_stopper[1].retract
        OnMouseDown: execute { dIO_LC.valve_stopper[1].extend := FALSE; dIO_LC.valve_stopper[1].retract := TRUE; }
    Lamp1 (1797,275 30x30), variable: dIO_LC.valve_stopper[1].extended, style: Lamp-Lamp1-Green
    Lamp1 (1799,351 30x30), variable: dIO_LC.valve_stopper[1].retracted, style: Lamp-Lamp1-Green
    Label (1851,277 132x26), "extended"
    Label (1854,350 132x26), "retracted"
    Button (1653,434 93x52), "Extend", colour toggle: dIO_LC.valve_guide[0].extend
        OnMouseDown: execute { dIO_LC.valve_guide[0].extend := TRUE; dIO_LC.valve_guide[0].retract := FALSE; }
    Button (1654,510 93x52), "retract", colour toggle: dIO_LC.valve_guide[0].retract
        OnMouseDown: execute { dIO_LC.valve_guide[0].extend := FALSE; dIO_LC.valve_guide[0].retract := TRUE; }
    Lamp1 (1798,447 30x30), variable: dIO_LC.valve_guide[0].extended, style: Lamp-Lamp1-Green
    Lamp1 (1800,523 30x30), variable: dIO_LC.valve_guide[0].retracted, style: Lamp-Lamp1-Green
    Label (1852,449 132x26), "extended"
    Label (1855,522 132x26), "retracted"
    Button (1645,610 93x52), "Extend", colour toggle: dIO_LC.valve_guide[1].extend
        OnMouseDown: execute { dIO_LC.valve_guide[1].extend := TRUE; dIO_LC.valve_guide[1].retract := FALSE; }
    Button (1646,686 93x52), "retract", colour toggle: dIO_LC.valve_guide[1].retract
        OnMouseDown: execute { dIO_LC.valve_guide[1].extend := FALSE; dIO_LC.valve_guide[1].retract := TRUE; }
    Lamp1 (1790,623 30x30), variable: dIO_LC.valve_guide[1].extended, style: Lamp-Lamp1-Green
    Lamp1 (1792,699 30x30), variable: dIO_LC.valve_guide[1].retracted, style: Lamp-Lamp1-Green
    Label (1844,625 132x26), "extended"
    Label (1847,698 132x26), "retracted"
    Lamp1 (978,921 30x30), variable: dIO_LC.pressure_sensor, style: Lamp-Lamp1-Green
    Label (1032,923 132x26), "air pressure"
END_VISUALIZATION

// ---- VISUs/v_LB.TcVIS
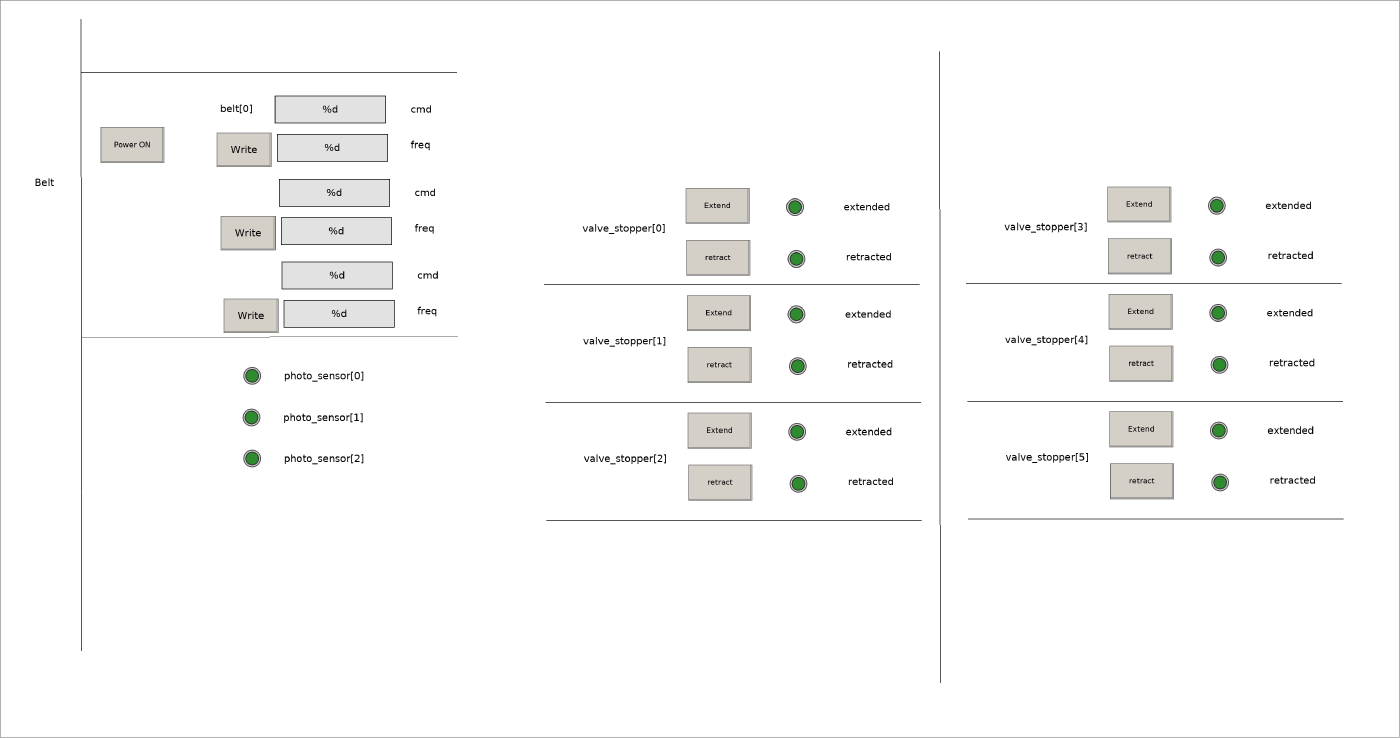
VISUALIZATION v_LB  // 2048x1080
VAR_IN_OUT
	dIO_LB		: LateralBuf_Module;
END_VAR
    Line (118,28) (119,952)
    Line (119,106) (668,106)
    Label (833,321 160x26), "valve_stopper[0]"
    Button (1003,275 93x52), "Extend", colour toggle: dIO_LB.valve_stopper[0].extend
        OnMouseDown: execute { dIO_LB.valve_stopper[0].extend := TRUE; dIO_LB.valve_stopper[0].retract := FALSE; }
    Button (1004,351 93x52), "retract", colour toggle: dIO_LB.valve_stopper[0].retract
        OnMouseDown: execute { dIO_LB.valve_stopper[0].extend := FALSE; dIO_LB.valve_stopper[0].retract := TRUE; }
    Lamp1 (1148,288 30x30), variable: dIO_LB.valve_stopper[0].extended, style: Lamp-Lamp1-Green
    Lamp1 (1150,364 30x30), variable: dIO_LB.valve_stopper[0].retracted, style: Lamp-Lamp1-Green
    Label (1202,290 132x26), "extended"
    Label (1205,363 132x26), "retracted"
    Label (834,486 160x26), "valve_stopper[1]"
    Line (796,416) (1345,416)
    Line (798,589) (1347,589)
    Rectangle (402,140 162x40), "%d", text variable: dIO_LB.belt[0].fbconverter.cmd
        OnMouseClick: write the text variable via Default
    Rectangle (405,196 162x40), "%d", text variable: dIO_LB.belt[0].fbconverter.freq
        OnMouseClick: write the text variable via Default
    Label (280,146 132x26), "belt[0]"
    Label (550,147 132x26), "cmd"
    Label (549,199 132x26), "freq"
    Button (147,186 93x52), "Power ON", colour toggle: dIO_LB.power_beltConv
        toggle dIO_LB.power_beltConv
    Button (317,194 80x50), "Write"
        OnMouseDown: execute { dIO_LB.belt[0].fbconverter.bSetParaEx	:= TRUE; }
        OnMouseUp: execute { dIO_LB.belt[0].fbconverter.bSetParaEx	:= FALSE; }
    Lamp1 (354,535 30x30), variable: dIO_LB.photo_sensor[0], style: Lamp-Lamp1-Green
    Label (408,537 132x26), "photo_sensor[0]"
    Lamp1 (353,596 30x30), variable: dIO_LB.photo_sensor[1], style: Lamp-Lamp1-Green
    Label (407,598 132x26), "photo_sensor[1]"
    Lamp1 (354,656 30x30), variable: dIO_LB.photo_sensor[2], style: Lamp-Lamp1-Green
    Label (408,658 132x26), "photo_sensor[2]"
    Line (120,493) (669,492)
    Label (25,254 80x26), "Belt"
    Button (1005,432 93x52), "Extend", colour toggle: dIO_LB.valve_stopper[1].extend
        OnMouseDown: execute { dIO_LB.valve_stopper[1].extend := TRUE; dIO_LB.valve_stopper[1].retract := FALSE; }
    Button (1006,508 93x52), "retract", colour toggle: dIO_LB.valve_stopper[1].retract
        OnMouseDown: execute { dIO_LB.valve_stopper[1].extend := FALSE; dIO_LB.valve_stopper[1].retract := TRUE; }
    Lamp1 (1150,445 30x30), variable: dIO_LB.valve_stopper[1].extended, style: Lamp-Lamp1-Green
    Lamp1 (1152,521 30x30), variable: dIO_LB.valve_stopper[1].retracted, style: Lamp-Lamp1-Green
    Label (1204,447 132x26), "extended"
    Label (1207,520 132x26), "retracted"
    Rectangle (408,262 162x40), "%d", text variable: dIO_LB.belt[1].fbconverter.cmd
        OnMouseClick: write the text variable via Default
    Rectangle (411,318 162x40), "%d", text variable: dIO_LB.belt[1].fbconverter.freq
        OnMouseClick: write the text variable via Default
    Label (556,269 132x26), "cmd"
    Label (555,321 132x26), "freq"
    Button (323,316 80x50), "Write"
        OnMouseDown: execute { dIO_LB.belt[1].fbconverter.bSetParaEx	:= TRUE; }
        OnMouseUp: execute { dIO_LB.belt[1].fbconverter.bSetParaEx	:= FALSE; }
    Rectangle (412,383 162x40), "%d", text variable: dIO_LB.belt[2].fbconverter.cmd
        OnMouseClick: write the text variable via Default
    Rectangle (415,439 162x40), "%d", text variable: dIO_LB.belt[2].fbconverter.freq
        OnMouseClick: write the text variable via Default
    Label (560,390 132x26), "cmd"
    Label (559,442 132x26), "freq"
    Button (327,437 80x50), "Write"
        OnMouseDown: execute { dIO_LB.belt[2].fbconverter.bSetParaEx	:= TRUE; }
        OnMouseUp: execute { dIO_LB.belt[2].fbconverter.bSetParaEx	:= FALSE; }
    Label (835,658 160x26), "valve_stopper[2]"
    Line (799,761) (1348,761)
    Button (1006,604 93x52), "Extend", colour toggle: dIO_LB.valve_stopper[2].extend
        OnMouseDown: execute { dIO_LB.valve_stopper[2].extend := TRUE; dIO_LB.valve_stopper[2].retract := FALSE; }
    Button (1007,680 93x52), "retract", colour toggle: dIO_LB.valve_stopper[2].retract
        OnMouseDown: execute { dIO_LB.valve_stopper[2].extend := FALSE; dIO_LB.valve_stopper[2].retract := TRUE; }
    Lamp1 (1151,617 30x30), variable: dIO_LB.valve_stopper[2].extended, style: Lamp-Lamp1-Green
    Lamp1 (1153,693 30x30), variable: dIO_LB.valve_stopper[2].retracted, style: Lamp-Lamp1-Green
    Label (1205,619 132x26), "extended"
    Label (1208,692 132x26), "retracted"
    Label (1450,319 160x26), "valve_stopper[3]"
    Button (1620,273 93x52), "Extend", colour toggle: dIO_LB.valve_stopper[3].extend
        OnMouseDown: execute { dIO_LB.valve_stopper[3].extend := TRUE; dIO_LB.valve_stopper[3].retract := FALSE; }
    Button (1621,349 93x52), "retract", colour toggle: dIO_LB.valve_stopper[3].retract
        OnMouseDown: execute { dIO_LB.valve_stopper[3].extend := FALSE; dIO_LB.valve_stopper[3].retract := TRUE; }
    Lamp1 (1765,286 30x30), variable: dIO_LB.valve_stopper[3].extended, style: Lamp-Lamp1-Green
    Lamp1 (1767,362 30x30), variable: dIO_LB.valve_stopper[3].retracted, style: Lamp-Lamp1-Green
    Label (1819,288 132x26), "extended"
    Label (1822,361 132x26), "retracted"
    Label (1451,484 160x26), "valve_stopper[4]"
    Line (1413,414) (1962,414)
    Line (1415,587) (1964,587)
    Button (1622,430 93x52), "Extend", colour toggle: dIO_LB.valve_stopper[4].extend
        OnMouseDown: execute { dIO_LB.valve_stopper[4].extend := TRUE; dIO_LB.valve_stopper[4].retract := FALSE; }
    Button (1623,506 93x52), "retract", colour toggle: dIO_LB.valve_stopper[4].retract
        OnMouseDown: execute { dIO_LB.valve_stopper[4].extend := FALSE; dIO_LB.valve_stopper[4].retract := TRUE; }
    Lamp1 (1767,443 30x30), variable: dIO_LB.valve_stopper[4].extended, style: Lamp-Lamp1-Green
    Lamp1 (1769,519 30x30), variable: dIO_LB.valve_stopper[4].retracted, style: Lamp-Lamp1-Green
    Label (1821,445 132x26), "extended"
    Label (1824,518 132x26), "retracted"
    Label (1452,656 160x26), "valve_stopper[5]"
    Line (1416,759) (1965,759)
    Button (1623,602 93x52), "Extend", colour toggle: dIO_LB.valve_stopper[5].extend
        OnMouseDown: execute { dIO_LB.valve_stopper[5].extend := TRUE; dIO_LB.valve_stopper[5].retract := FALSE; }
    Button (1624,678 93x52), "retract", colour toggle: dIO_LB.valve_stopper[5].retract
        OnMouseDown: execute { dIO_LB.valve_stopper[5].extend := FALSE; dIO_LB.valve_stopper[5].retract := TRUE; }
    Lamp1 (1768,615 30x30), variable: dIO_LB.valve_stopper[5].extended, style: Lamp-Lamp1-Green
    Lamp1 (1770,691 30x30), variable: dIO_LB.valve_stopper[5].retracted, style: Lamp-Lamp1-Green
    Label (1822,617 132x26), "extended"
    Label (1825,690 132x26), "retracted"
    Line (1374,75) (1375,999)
END_VISUALIZATION

// ---- VISUs/v_rem_0.TcVIS
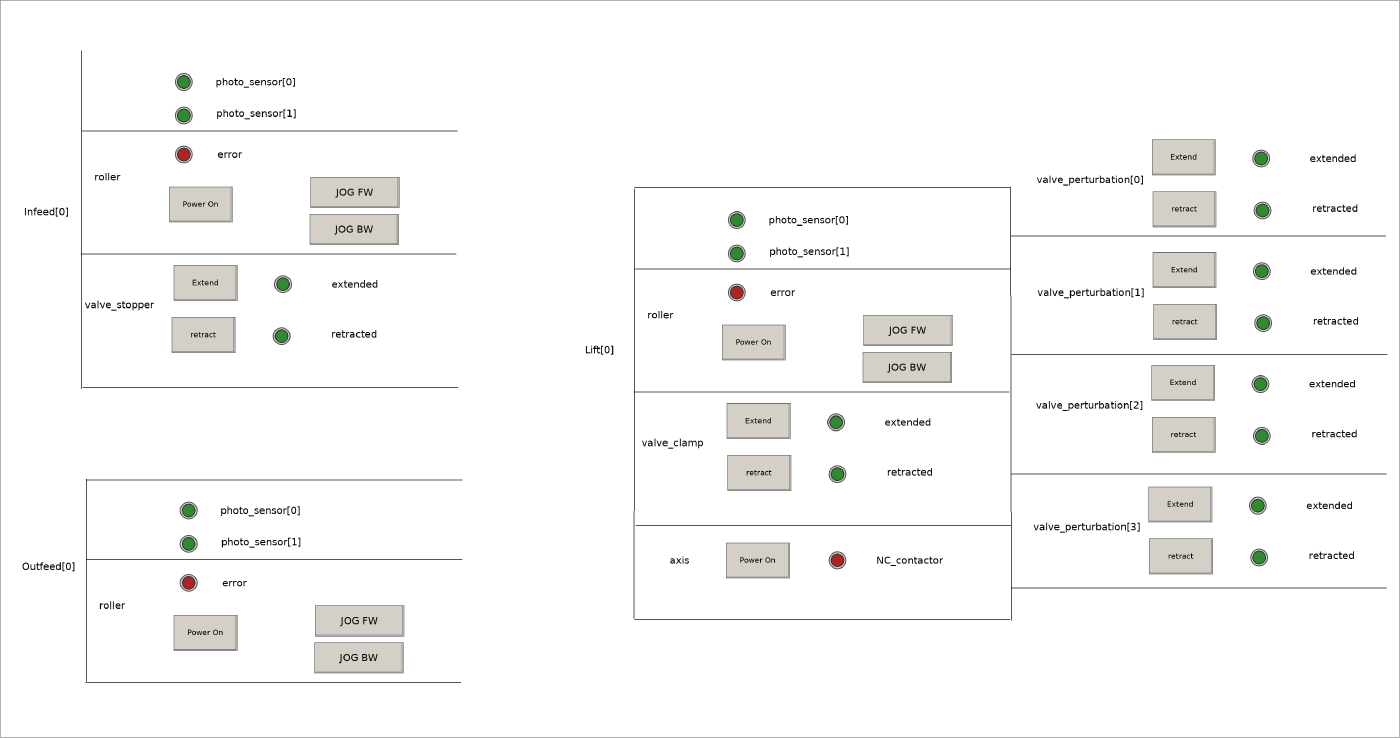
VISUALIZATION v_rem_0  // 2048x1080
VAR_IN_OUT
	dIO_ReM		: Replenishment_Module;
END_VAR
    Lamp1 (254,105 30x30), variable: dIO_ReM.infeed[0].photo_sensor[0].debounced_input.Q, style: Lamp-Lamp1-Green
    Lamp1 (254,154 30x30), variable: dIO_ReM.infeed[0].photo_sensor[1].debounced_input.Q, style: Lamp-Lamp1-Green
    Label (308,107 132x26), "photo_sensor[0]"
    Label (309,153 132x26), "photo_sensor[1]"
    Label (28,297 80x26), "Infeed[0]"
    Lamp1 (254,211 30x30), variable: dIO_ReM.infeed[0].roller.err, style: Lamp-Lamp1-Red
    Label (270,213 132x26), "error"
    Label (91,246 132x26), "roller"
    Line (120,191) (669,191)
    Line (119,74) (119,569)
    Label (109,433 132x26), "valve_stopper"
    Button (454,259 130x45), "JOG FW", colour toggle: dIO_ReM.infeed[0].roller.forward
        OnMouseDown: execute { dIO_ReM.infeed[0].roller.forward := TRUE; }
        OnMouseUp: execute { dIO_ReM.infeed[0].roller.forward := FALSE; }
    Button (453,313 130x45), "JOG BW", colour toggle: dIO_ReM.infeed[0].roller.backward
        OnMouseDown: execute { dIO_ReM.infeed[0].roller.backward := TRUE; }
        OnMouseUp: execute { dIO_ReM.infeed[0].roller.backward := FALSE; }
    Button (247,273 93x52), "Power On", colour toggle: dIO_ReM.infeed[0].roller.Power
        toggle dIO_ReM.infeed[0].roller.Power
    Button (254,388 93x52), "Extend", colour toggle: dIO_ReM.infeed[0].valve_stopper.extend
        OnMouseDown: execute { dIO_ReM.infeed[0].valve_stopper.extend := TRUE; dIO_ReM.infeed[0].valve_stopper.retract := FALSE; }
    Button (251,464 93x52), "retract", colour toggle: dIO_ReM.infeed[0].valve_stopper.retract
        OnMouseDown: execute { dIO_ReM.infeed[0].valve_stopper.extend := FALSE; dIO_ReM.infeed[0].valve_stopper.retract := TRUE; }
    Lamp1 (399,401 30x30), variable: dIO_ReM.infeed[0].valve_stopper.extended, style: Lamp-Lamp1-Green
    Lamp1 (397,477 30x30), variable: dIO_ReM.infeed[0].valve_stopper.retracted, style: Lamp-Lamp1-Green
    Label (453,403 132x26), "extended"
    Label (452,476 132x26), "retracted"
    Line (118,371) (667,371)
    Line (121,567) (670,567)
    Lamp1 (261,732 30x30), variable: dIO_ReM.outfeed[0].photo_sensor[0].debounced_input.Q, style: Lamp-Lamp1-Green
    Lamp1 (261,781 30x30), variable: dIO_ReM.outfeed[0].photo_sensor[1].debounced_input.Q, style: Lamp-Lamp1-Green
    Label (315,734 132x26), "photo_sensor[0]"
    Label (316,780 132x26), "photo_sensor[1]"
    Label (31,816 80x26), "Outfeed[0]"
    Lamp1 (261,838 30x30), variable: dIO_ReM.outfeed[0].roller.err, style: Lamp-Lamp1-Red
    Label (277,840 132x26), "error"
    Label (98,873 132x26), "roller"
    Line (127,818) (676,818)
    Line (126,701) (126,997)
    Button (461,886 130x45), "JOG FW", colour toggle: dIO_ReM.outfeed[0].roller.forward
        OnMouseDown: execute { dIO_ReM.outfeed[0].roller.forward := TRUE; }
        OnMouseUp: execute { dIO_ReM.outfeed[0].roller.forward := FALSE; }
    Button (460,940 130x45), "JOG BW", colour toggle: dIO_ReM.outfeed[0].roller.backward
        OnMouseDown: execute { dIO_ReM.outfeed[0].roller.backward := TRUE; }
        OnMouseUp: execute { dIO_ReM.outfeed[0].roller.backward := FALSE; }
    Button (254,900 93x52), "Power On", colour toggle: dIO_ReM.outfeed[0].roller.Power
        toggle dIO_ReM.outfeed[0].roller.Power
    Line (125,998) (674,998)
    Line (127,702) (676,702)
    Lamp1 (1063,307 30x30), variable: dIO_ReM.lift[0].photo_sensor[0].debounced_input.Q, style: Lamp-Lamp1-Green
    Lamp1 (1063,356 30x30), variable: dIO_ReM.lift[0].photo_sensor[1].debounced_input.Q, style: Lamp-Lamp1-Green
    Label (1117,309 132x26), "photo_sensor[0]"
    Label (1118,355 132x26), "photo_sensor[1]"
    Label (837,499 80x26), "Lift[0]"
    Lamp1 (1063,413 30x30), variable: dIO_ReM.lift[0].roller.err, style: Lamp-Lamp1-Red
    Label (1079,415 132x26), "error"
    Label (900,448 132x26), "roller"
    Line (929,393) (1478,393)
    Line (928,276) (927,905)
    Label (918,635 132x26), "valve_clamp"
    Button (1263,461 130x45), "JOG FW", colour toggle: dIO_ReM.lift[0].roller.forward
        OnMouseDown: execute { dIO_ReM.lift[0].roller.forward := TRUE; }
        OnMouseUp: execute { dIO_ReM.lift[0].roller.forward := FALSE; }
    Button (1262,515 130x45), "JOG BW", colour toggle: dIO_ReM.lift[0].roller.backward
        OnMouseDown: execute { dIO_ReM.lift[0].roller.backward := TRUE; }
        OnMouseUp: execute { dIO_ReM.lift[0].roller.backward := FALSE; }
    Button (1056,475 93x52), "Power On", colour toggle: dIO_ReM.lift[0].roller.Power
        toggle dIO_ReM.lift[0].roller.Power
    Button (1063,590 93x52), "Extend", colour toggle: dIO_ReM.lift[0].valve_clamp.extend
        OnMouseDown: execute { dIO_ReM.lift[0].valve_clamp.extend := TRUE; dIO_ReM.lift[0].valve_clamp.retract := FALSE; }
    Button (1064,666 93x52), "retract", colour toggle: dIO_ReM.lift[0].valve_clamp.retract
        OnMouseDown: execute { dIO_ReM.lift[0].valve_clamp.extend := FALSE; dIO_ReM.lift[0].valve_clamp.retract := TRUE; }
    Lamp1 (1208,603 30x30), variable: dIO_ReM.lift[0].valve_clamp.extended, style: Lamp-Lamp1-Green
    Lamp1 (1210,679 30x30), variable: dIO_ReM.lift[0].valve_clamp.retracted, style: Lamp-Lamp1-Green
    Label (1262,605 132x26), "extended"
    Label (1265,678 132x26), "retracted"
    Line (927,573) (1476,573)
    Line (930,769) (1479,769)
    Label (1515,250 160x26), "valve_perturbation[0]"
    Button (1685,204 93x52), "Extend", colour toggle: dIO_ReM.lift[0].valve_perturbation[0].extend
        OnMouseDown: execute { dIO_ReM.lift[0].valve_perturbation[0].extend := TRUE; dIO_ReM.lift[0].valve_perturbation[0].retract := FALSE; }
    Button (1686,280 93x52), "retract", colour toggle: dIO_ReM.lift[0].valve_perturbation[0].retract
        OnMouseDown: execute { dIO_ReM.lift[0].valve_perturbation[0].extend := FALSE; dIO_ReM.lift[0].valve_perturbation[0].retract := TRUE; }
    Lamp1 (1830,217 30x30), variable: dIO_ReM.lift[0].valve_perturbation[0].extended, style: Lamp-Lamp1-Green
    Lamp1 (1832,293 30x30), variable: dIO_ReM.lift[0].valve_perturbation[0].retracted, style: Lamp-Lamp1-Green
    Label (1884,219 132x26), "extended"
    Label (1887,292 132x26), "retracted"
    Label (1516,415 160x26), "valve_perturbation[1]"
    Button (1686,369 93x52), "Extend", colour toggle: dIO_ReM.lift[0].valve_perturbation[1].extend
        OnMouseDown: execute { dIO_ReM.lift[0].valve_perturbation[1].extend := TRUE; dIO_ReM.lift[0].valve_perturbation[1].retract := FALSE; }
    Button (1687,445 93x52), "retract", colour toggle: dIO_ReM.lift[0].valve_perturbation[1].retract
        OnMouseDown: execute { dIO_ReM.lift[0].valve_perturbation[1].extend := FALSE; dIO_ReM.lift[0].valve_perturbation[1].retract := TRUE; }
    Lamp1 (1831,382 30x30), variable: dIO_ReM.lift[0].valve_perturbation[1].extended, style: Lamp-Lamp1-Green
    Lamp1 (1833,458 30x30), variable: dIO_ReM.lift[0].valve_perturbation[1].retracted, style: Lamp-Lamp1-Green
    Label (1885,384 132x26), "extended"
    Label (1888,457 132x26), "retracted"
    Label (1514,580 160x26), "valve_perturbation[2]"
    Button (1684,534 93x52), "Extend", colour toggle: dIO_ReM.lift[0].valve_perturbation[2].extend
        OnMouseDown: execute { dIO_ReM.lift[0].valve_perturbation[2].extend := TRUE; dIO_ReM.lift[0].valve_perturbation[2].retract := FALSE; }
    Button (1685,610 93x52), "retract", colour toggle: dIO_ReM.lift[0].valve_perturbation[2].retract
        OnMouseDown: execute { dIO_ReM.lift[0].valve_perturbation[2].extend := FALSE; dIO_ReM.lift[0].valve_perturbation[2].retract := TRUE; }
    Lamp1 (1829,547 30x30), variable: dIO_ReM.lift[0].valve_perturbation[2].extended, style: Lamp-Lamp1-Green
    Lamp1 (1831,623 30x30), variable: dIO_ReM.lift[0].valve_perturbation[2].retracted, style: Lamp-Lamp1-Green
    Label (1883,549 132x26), "extended"
    Label (1886,622 132x26), "retracted"
    Label (1510,758 160x26), "valve_perturbation[3]"
    Button (1680,712 93x52), "Extend", colour toggle: dIO_ReM.lift[0].valve_perturbation[3].extend
        OnMouseDown: execute { dIO_ReM.lift[0].valve_perturbation[3].extend := TRUE; dIO_ReM.lift[0].valve_perturbation[3].retract := FALSE; }
    Button (1681,788 93x52), "retract", colour toggle: dIO_ReM.lift[0].valve_perturbation[3].retract
        OnMouseDown: execute { dIO_ReM.lift[0].valve_perturbation[3].extend := FALSE; dIO_ReM.lift[0].valve_perturbation[3].retract := TRUE; }
    Lamp1 (1825,725 30x30), variable: dIO_ReM.lift[0].valve_perturbation[3].extended, style: Lamp-Lamp1-Green
    Lamp1 (1827,801 30x30), variable: dIO_ReM.lift[0].valve_perturbation[3].retracted, style: Lamp-Lamp1-Green
    Label (1879,727 132x26), "extended"
    Label (1882,800 132x26), "retracted"
    Line (1478,273) (1479,908)
    Line (1478,345) (2027,345)
    Line (1480,518) (2029,518)
    Line (1479,693) (2028,693)
    Line (1479,860) (2028,860)
    Line (928,274) (1477,274)
    Line (928,906) (1477,906)
    Label (1265,807 132x26), "NC_contactor"
    Label (928,807 132x26), "axis"
    Button (1062,794 93x52), "Power On", colour toggle: dIO_ReM.lift[0].power_axis
        toggle dIO_ReM.lift[0].power_axis
    Lamp1 (1210,805 30x30), variable: dIO_ReM.lift[0].contactor_axis, style: Lamp-Lamp1-Red
END_VISUALIZATION

// ---- VISUs/v_pm_0.TcVIS
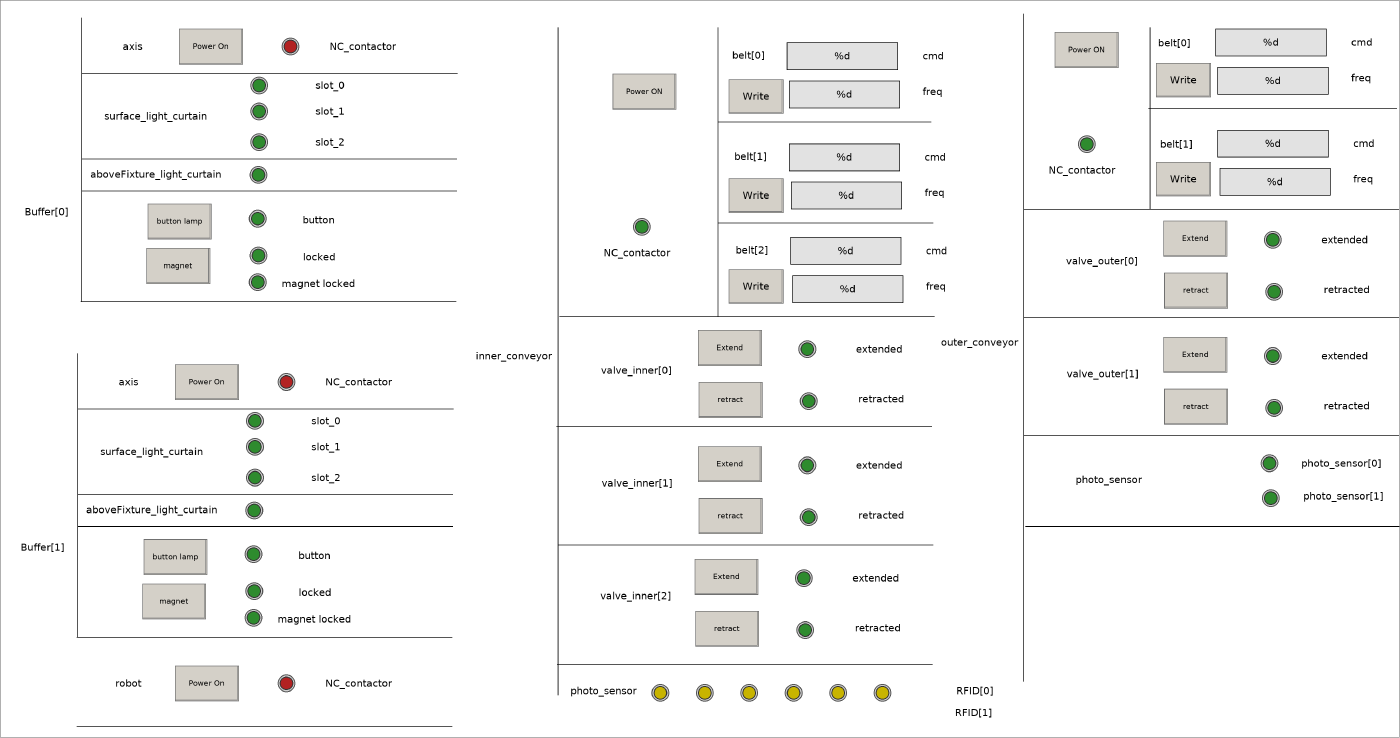
VISUALIZATION v_pm_0  // 2048x1080
VAR_IN_OUT
	dIO_PM		: Picking_Module;
END_VAR
    Lamp1 (364,110 30x30), variable: dIO_PM.buffer[0].surfae_slot_0, style: Lamp-Lamp1-Green
    Label (418,112 130x26), "slot_0"
    Label (28,297 80x26), "Buffer[0]"
    Line (120,107) (669,107)
    Line (119,26) (119,441)
    Line (118,441) (667,441)
    Label (672,508 160x26), "inner_conveyor"
    Line (816,40) (816,1017)
    Label (851,529 160x26), "valve_inner[0]"
    Button (1021,483 93x52), "Extend", colour toggle: dIO_PM.inConv.valve[0].extend
        OnMouseDown: execute { dIO_PM.inConv.valve[0].extend := TRUE; dIO_PM.inConv.valve[0].retract := FALSE; }
    Button (1022,559 93x52), "retract", colour toggle: dIO_PM.inConv.valve[0].retract
        OnMouseDown: execute { dIO_PM.inConv.valve[0].extend := FALSE; dIO_PM.inConv.valve[0].retract := TRUE; }
    Lamp1 (1166,496 30x30), variable: dIO_PM.inConv.valve[0].extended, style: Lamp-Lamp1-Green
    Lamp1 (1168,572 30x30), variable: dIO_PM.inConv.valve[0].retracted, style: Lamp-Lamp1-Green
    Label (1220,498 132x26), "extended"
    Label (1223,571 132x26), "retracted"
    Label (852,694 160x26), "valve_inner[1]"
    Label (850,859 160x26), "valve_inner[2]"
    Line (814,624) (1363,624)
    Line (816,797) (1365,797)
    Line (815,972) (1364,972)
    Label (465,55 132x26), "NC_contactor"
    Label (128,55 132x26), "axis"
    Button (262,42 93x52), "Power On", colour toggle: dIO_PM.buffer[0].power_axis
        toggle dIO_PM.buffer[0].power_axis
    Lamp1 (410,53 30x30), variable: dIO_PM.buffer[0].contractor_axis, style: Lamp-Lamp1-Red
    Label (128,157 200x26), "surface_light_curtain"
    Label (418,150 130x26), "slot_1"
    Lamp1 (364,148 30x30), variable: dIO_PM.buffer[0].surfae_slot_1, style: Lamp-Lamp1-Green
    Label (418,195 130x26), "slot_2"
    Lamp1 (364,193 30x30), variable: dIO_PM.buffer[0].surfae_slot_2, style: Lamp-Lamp1-Green
    Label (128,242 200x26), "aboveFixture_light_curtain"
    Lamp1 (363,241 30x30), variable: dIO_PM.buffer[0].above_fixture_light_curtain, style: Lamp-Lamp1-Green
    Line (119,232) (668,232)
    Line (119,279) (668,279)
    Label (406,309 120x26), "button"
    Lamp1 (362,305 30x30), variable: dIO_PM.buffer[0].button, style: Lamp-Lamp1-Green
    Button (216,298 93x52), "button lamp", colour toggle: dIO_PM.buffer[0].lamp_button
        toggle dIO_PM.buffer[0].lamp_button
    Button (214,363 93x52), "magnet", colour toggle: dIO_PM.buffer[0].magnet
        toggle dIO_PM.buffer[0].magnet
    Label (407,363 120x26), "locked"
    Lamp1 (363,359 30x30), variable: dIO_PM.buffer[0].locked, style: Lamp-Lamp1-Green
    Label (406,402 120x26), "magnet locked"
    Lamp1 (362,398 30x30), variable: dIO_PM.buffer[0].magnet_locked, style: Lamp-Lamp1-Green
    Lamp1 (358,601 30x30), variable: dIO_PM.buffer[1].surfae_slot_0, style: Lamp-Lamp1-Green
    Label (412,603 130x26), "slot_0"
    Label (22,788 80x26), "Buffer[1]"
    Line (114,598) (663,598)
    Line (113,517) (113,932)
    Line (112,932) (661,932)
    Label (459,546 132x26), "NC_contactor"
    Label (122,546 132x26), "axis"
    Button (256,533 93x52), "Power On", colour toggle: dIO_PM.buffer[1].power_axis
        toggle dIO_PM.buffer[1].power_axis
    Lamp1 (404,544 30x30), variable: dIO_PM.buffer[1].contractor_axis, style: Lamp-Lamp1-Red
    Label (122,648 200x26), "surface_light_curtain"
    Label (412,641 130x26), "slot_1"
    Lamp1 (358,639 30x30), variable: dIO_PM.buffer[1].surfae_slot_1, style: Lamp-Lamp1-Green
    Label (412,686 130x26), "slot_2"
    Lamp1 (358,684 30x30), variable: dIO_PM.buffer[1].surfae_slot_2, style: Lamp-Lamp1-Green
    Label (122,733 200x26), "aboveFixture_light_curtain"
    Lamp1 (357,732 30x30), variable: dIO_PM.buffer[1].above_fixture_light_curtain, style: Lamp-Lamp1-Green
    Line (113,723) (662,723)
    Line (113,770) (662,770)
    Label (400,800 120x26), "button"
    Lamp1 (356,796 30x30), variable: dIO_PM.buffer[1].button, style: Lamp-Lamp1-Green
    Button (210,789 93x52), "button lamp", colour toggle: dIO_PM.buffer[1].lamp_button
        toggle dIO_PM.buffer[1].lamp_button
    Button (208,854 93x52), "magnet", colour toggle: dIO_PM.buffer[1].magnet
        toggle dIO_PM.buffer[1].magnet
    Label (401,854 120x26), "locked"
    Lamp1 (357,850 30x30), variable: dIO_PM.buffer[1].locked, style: Lamp-Lamp1-Green
    Label (400,893 120x26), "magnet locked"
    Lamp1 (356,889 30x30), variable: dIO_PM.buffer[1].magnet_locked, style: Lamp-Lamp1-Green
    Line (112,1063) (661,1063)
    Label (459,987 132x26), "NC_contactor"
    Label (122,987 132x26), "robot"
    Button (256,974 93x52), "Power On", colour toggle: dIO_PM.power_robot
        toggle dIO_PM.power_robot
    Lamp1 (404,985 30x30), variable: dIO_PM.contactor_robot, style: Lamp-Lamp1-Red
    Rectangle (1151,62 162x40), "%d", text variable: dIO_PM.inConv.belt[0].fbconverter.cmd
        OnMouseClick: write the text variable via Default
    Rectangle (1154,118 162x40), "%d", text variable: dIO_PM.inConv.belt[0].fbconverter.freq
        OnMouseClick: write the text variable via Default
    Label (1029,68 132x26), "belt[0]"
    Label (1299,69 132x26), "cmd"
    Label (1298,121 132x26), "freq"
    Line (1050,178) (1362,178)
    Rectangle (1154,210 162x40), "%d", text variable: dIO_PM.inConv.belt[1].fbconverter.cmd
        OnMouseClick: write the text variable via Default
    Rectangle (1157,266 162x40), "%d", text variable: dIO_PM.inConv.belt[1].fbconverter.freq
        OnMouseClick: write the text variable via Default
    Label (1032,216 132x26), "belt[1]"
    Label (1302,217 132x26), "cmd"
    Label (1301,269 132x26), "freq"
    Line (1050,326) (1365,326)
    Rectangle (1156,347 162x40), "%d", text variable: dIO_PM.inConv.belt[2].fbconverter.cmd
        OnMouseClick: write the text variable via Default
    Rectangle (1159,403 162x40), "%d", text variable: dIO_PM.inConv.belt[2].fbconverter.freq
        OnMouseClick: write the text variable via Default
    Label (1034,353 132x26), "belt[2]"
    Label (1304,354 132x26), "cmd"
    Label (1303,406 132x26), "freq"
    Line (818,463) (1367,463)
    Button (1021,653 93x52), "Extend", colour toggle: dIO_PM.inConv.valve[1].extend
        OnMouseDown: execute { dIO_PM.inConv.valve[1].extend := TRUE; dIO_PM.inConv.valve[1].retract := FALSE; }
    Button (1022,729 93x52), "retract", colour toggle: dIO_PM.inConv.valve[1].retract
        OnMouseDown: execute { dIO_PM.inConv.valve[1].extend := FALSE; dIO_PM.inConv.valve[1].retract := TRUE; }
    Lamp1 (1166,666 30x30), variable: dIO_PM.inConv.valve[1].extended, style: Lamp-Lamp1-Green
    Lamp1 (1168,742 30x30), variable: dIO_PM.inConv.valve[1].retracted, style: Lamp-Lamp1-Green
    Label (1220,668 132x26), "extended"
    Label (1223,741 132x26), "retracted"
    Button (1016,818 93x52), "Extend", colour toggle: dIO_PM.inConv.valve[2].extend
        OnMouseDown: execute { dIO_PM.inConv.valve[2].extend := TRUE; dIO_PM.inConv.valve[2].retract := FALSE; }
    Button (1017,894 93x52), "retract", colour toggle: dIO_PM.inConv.valve[2].retract
        OnMouseDown: execute { dIO_PM.inConv.valve[2].extend := FALSE; dIO_PM.inConv.valve[2].retract := TRUE; }
    Lamp1 (1161,831 30x30), variable: dIO_PM.inConv.valve[2].extended, style: Lamp-Lamp1-Green
    Lamp1 (1163,907 30x30), variable: dIO_PM.inConv.valve[2].retracted, style: Lamp-Lamp1-Green
    Label (1215,833 132x26), "extended"
    Label (1218,906 132x26), "retracted"
    Label (1346,998 160x26), "RFID[0]"
    Label (1344,1030 160x26), "RFID[1]"
    Label (1353,488 160x26), "outer_conveyor"
    Line (1497,20) (1497,997)
    Label (1532,369 160x26), "valve_outer[0]"
    Button (1702,323 93x52), "Extend", colour toggle: dIO_PM.outConv.valve[0].extend
        OnMouseDown: execute { dIO_PM.outConv.valve[0].extend := TRUE; dIO_PM.outConv.valve[0].retract := FALSE; }
    Button (1703,399 93x52), "retract", colour toggle: dIO_PM.outConv.valve[0].retract
        OnMouseDown: execute { dIO_PM.outConv.valve[0].extend := FALSE; dIO_PM.outConv.valve[0].retract := TRUE; }
    Lamp1 (1847,336 30x30), variable: dIO_PM.outConv.valve[0].extended, style: Lamp-Lamp1-Green
    Lamp1 (1849,412 30x30), variable: dIO_PM.outConv.valve[0].retracted, style: Lamp-Lamp1-Green
    Label (1901,338 132x26), "extended"
    Label (1904,411 132x26), "retracted"
    Label (1533,534 160x26), "valve_outer[1]"
    Line (1498,464) (2047,464)
    Line (1497,637) (2046,637)
    Line (1500,770) (2049,770)
    Rectangle (1778,42 162x40), "%d", text variable: dIO_PM.outConv.belt[0].fbconverter.cmd
        OnMouseClick: write the text variable via Default
    Rectangle (1781,98 162x40), "%d", text variable: dIO_PM.outConv.belt[0].fbconverter.freq
        OnMouseClick: write the text variable via Default
    Label (1652,50 132x26), "belt[0]"
    Label (1926,49 132x26), "cmd"
    Label (1925,101 132x26), "freq"
    Line (1680,158) (2043,158)
    Rectangle (1781,190 162x40), "%d", text variable: dIO_PM.outConv.belt[1].fbconverter.cmd
        OnMouseClick: write the text variable via Default
    Rectangle (1784,246 162x40), "%d", text variable: dIO_PM.outConv.belt[1].fbconverter.freq
        OnMouseClick: write the text variable via Default
    Label (1655,198 132x26), "belt[1]"
    Label (1929,197 132x26), "cmd"
    Label (1928,249 132x26), "freq"
    Line (1497,306) (2046,306)
    Button (1702,493 93x52), "Extend", colour toggle: dIO_PM.outConv.valve[1].extend
        OnMouseDown: execute { dIO_PM.outConv.valve[1].extend := TRUE; dIO_PM.outConv.valve[1].retract := FALSE; }
    Button (1703,569 93x52), "retract", colour toggle: dIO_PM.outConv.valve[1].retract
        OnMouseDown: execute { dIO_PM.outConv.valve[1].extend := FALSE; dIO_PM.outConv.valve[1].retract := TRUE; }
    Lamp1 (1847,506 30x30), variable: dIO_PM.outConv.valve[1].extended, style: Lamp-Lamp1-Green
    Lamp1 (1849,582 30x30), variable: dIO_PM.outConv.valve[1].retracted, style: Lamp-Lamp1-Green
    Label (1901,508 132x26), "extended"
    Label (1904,581 132x26), "retracted"
    Lamp1 (1842,663 30x30), variable: dIO_PM.outConv.photo_sensor[0], style: Lamp-Lamp1-Green
    Lamp1 (1844,714 30x30), variable: dIO_PM.outConv.photo_sensor[1], style: Lamp-Lamp1-Green
    Label (1896,665 132x26), "photo_sensor[0]"
    Label (1899,713 132x26), "photo_sensor[1]"
    Label (1542,689 160x26), "photo_sensor"
    Line (1050,40) (1050,463)
    Button (896,108 93x52), "Power ON", colour toggle: dIO_PM.power_inConv
        toggle dIO_PM.power_inConv
    Lamp1 (924,317 30x30), variable: dIO_PM.contactor_inConv, style: Lamp-Lamp1-Green
    Label (866,357 132x26), "NC_contactor"
    Line (1682,40) (1682,306)
    Button (1543,47 93x52), "Power ON", colour toggle: dIO_PM.power_outConv
        toggle dIO_PM.power_outConv
    Lamp1 (1575,196 30x30), variable: dIO_PM.contactor_outConv, style: Lamp-Lamp1-Green
    Label (1517,236 132x26), "NC_contactor"
    Button (1066,116 80x50), "Write"
        OnMouseDown: execute { dIO_PM.inConv.belt[0].fbconverter.bSetParaEx	:= TRUE; }
        OnMouseUp: execute { dIO_PM.inConv.belt[0].fbconverter.bSetParaEx	:= FALSE; }
    Button (1066,261 80x50), "Write"
        OnMouseDown: execute { dIO_PM.inConv.belt[1].fbconverter.bSetParaEx	:= TRUE; }
        OnMouseUp: execute { dIO_PM.inConv.belt[1].fbconverter.bSetParaEx	:= FALSE; }
    Button (1066,394 80x50), "Write"
        OnMouseDown: execute { dIO_PM.inConv.belt[2].fbconverter.bSetParaEx	:= TRUE; }
        OnMouseUp: execute { dIO_PM.inConv.belt[2].fbconverter.bSetParaEx	:= FALSE; }
    Button (1691,237 80x50), "Write"
        OnMouseDown: execute { dIO_PM.outConv.belt[1].fbconverter.bSetParaEx	:= TRUE; }
        OnMouseUp: execute { dIO_PM.outConv.belt[1].fbconverter.bSetParaEx	:= FALSE; }
    Button (1691,92 80x50), "Write"
        OnMouseDown: execute { dIO_PM.outConv.belt[0].fbconverter.bSetParaEx	:= TRUE; }
        OnMouseUp: execute { dIO_PM.outConv.belt[0].fbconverter.bSetParaEx	:= FALSE; }
    Lamp1 (951,999 30x30), variable: dIO_PM.inConv.photo_sensor[0], style: Lamp-Lamp1-Yellow
    Lamp1 (1016,999 30x30), variable: dIO_PM.inConv.photo_sensor[1], style: Lamp-Lamp1-Yellow
    Lamp1 (1081,999 30x30), variable: dIO_PM.inConv.photo_sensor[2], style: Lamp-Lamp1-Yellow
    Lamp1 (1146,999 30x30), variable: dIO_PM.inConv.photo_sensor[3], style: Lamp-Lamp1-Yellow
    Lamp1 (1211,999 30x30), variable: dIO_PM.inConv.photo_sensor[4], style: Lamp-Lamp1-Yellow
    Lamp1 (1276,999 30x30), variable: dIO_PM.inConv.photo_sensor[5], style: Lamp-Lamp1-Yellow
    Label (803,998 160x26), "photo_sensor"
END_VISUALIZATION

// ---- VISUs/v_rem_1.TcVIS
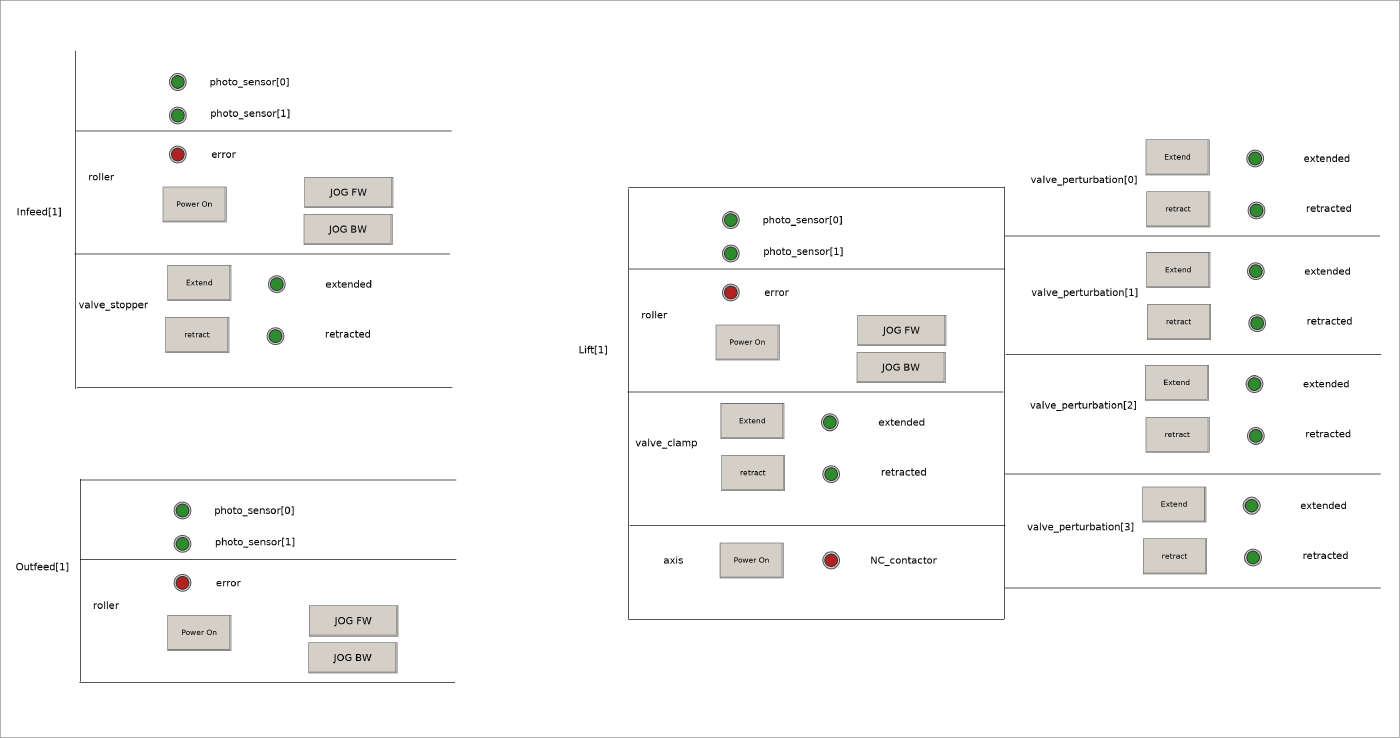
VISUALIZATION v_rem_1  // 2048x1080
VAR_IN_OUT
	dIO_ReM		: Replenishment_Module;
END_VAR
    Lamp1 (245,105 30x30), variable: dIO_ReM.infeed[1].photo_sensor[0].debounced_input.Q, style: Lamp-Lamp1-Green
    Lamp1 (245,154 30x30), variable: dIO_ReM.infeed[1].photo_sensor[1].debounced_input.Q, style: Lamp-Lamp1-Green
    Label (299,107 132x26), "photo_sensor[0]"
    Label (300,153 132x26), "photo_sensor[1]"
    Label (19,297 77x26), "Infeed[1]"
    Lamp1 (245,211 30x30), variable: dIO_ReM.infeed[1].roller.err, style: Lamp-Lamp1-Red
    Label (261,213 132x26), "error"
    Label (82,246 132x26), "roller"
    Line (111,191) (660,191)
    Line (110,74) (110,569)
    Label (100,433 132x26), "valve_stopper"
    Button (445,259 130x45), "JOG FW", colour toggle: dIO_ReM.infeed[1].roller.forward
        OnMouseDown: execute { dIO_ReM.infeed[1].roller.forward := TRUE; }
        OnMouseUp: execute { dIO_ReM.infeed[1].roller.forward := FALSE; }
    Button (444,313 130x45), "JOG BW", colour toggle: dIO_ReM.infeed[1].roller.backward
        OnMouseDown: execute { dIO_ReM.infeed[1].roller.backward := TRUE; }
        OnMouseUp: execute { dIO_ReM.infeed[1].roller.backward := FALSE; }
    Button (238,273 93x52), "Power On", colour toggle: dIO_ReM.infeed[1].roller.Power
        toggle dIO_ReM.infeed[1].roller.Power
    Button (245,388 93x52), "Extend", colour toggle: dIO_ReM.infeed[1].valve_stopper.extend
        OnMouseDown: execute { dIO_ReM.infeed[1].valve_stopper.extend := TRUE; dIO_ReM.infeed[1].valve_stopper.retract := FALSE; }
    Button (242,464 93x52), "retract", colour toggle: dIO_ReM.infeed[1].valve_stopper.retract
        OnMouseDown: execute { dIO_ReM.infeed[1].valve_stopper.extend := FALSE; dIO_ReM.infeed[1].valve_stopper.retract := TRUE; }
    Lamp1 (390,401 30x30), variable: dIO_ReM.infeed[1].valve_stopper.extended, style: Lamp-Lamp1-Green
    Lamp1 (388,477 30x30), variable: dIO_ReM.infeed[1].valve_stopper.retracted, style: Lamp-Lamp1-Green
    Label (444,403 132x26), "extended"
    Label (443,476 132x26), "retracted"
    Line (109,371) (658,371)
    Line (112,567) (661,567)
    Lamp1 (252,732 30x30), variable: dIO_ReM.outfeed[1].photo_sensor[0].debounced_input.Q, style: Lamp-Lamp1-Green
    Lamp1 (252,781 30x30), variable: dIO_ReM.outfeed[1].photo_sensor[1].debounced_input.Q, style: Lamp-Lamp1-Green
    Label (306,734 132x26), "photo_sensor[0]"
    Label (307,780 132x26), "photo_sensor[1]"
    Label (22,816 80x27), "Outfeed[1]"
    Lamp1 (252,838 30x30), variable: dIO_ReM.outfeed[1].roller.err, style: Lamp-Lamp1-Red
    Label (268,840 132x26), "error"
    Label (89,873 132x26), "roller"
    Line (118,818) (667,818)
    Line (117,701) (117,997)
    Button (452,886 130x45), "JOG FW", colour toggle: dIO_ReM.outfeed[1].roller.forward
        OnMouseDown: execute { dIO_ReM.outfeed[1].roller.forward := TRUE; }
        OnMouseUp: execute { dIO_ReM.outfeed[1].roller.forward := FALSE; }
    Button (451,940 130x45), "JOG BW", colour toggle: dIO_ReM.outfeed[1].roller.backward
        OnMouseDown: execute { dIO_ReM.outfeed[1].roller.backward := TRUE; }
        OnMouseUp: execute { dIO_ReM.outfeed[1].roller.backward := FALSE; }
    Button (245,900 93x52), "Power On", colour toggle: dIO_ReM.outfeed[1].roller.Power
        toggle dIO_ReM.outfeed[1].roller.Power
    Line (116,998) (665,998)
    Line (118,702) (667,702)
    Lamp1 (1054,307 30x30), variable: dIO_ReM.lift[1].photo_sensor[0].debounced_input.Q, style: Lamp-Lamp1-Green
    Lamp1 (1054,356 30x30), variable: dIO_ReM.lift[1].photo_sensor[1].debounced_input.Q, style: Lamp-Lamp1-Green
    Label (1108,309 132x26), "photo_sensor[0]"
    Label (1109,355 132x26), "photo_sensor[1]"
    Label (828,499 80x26), "Lift[1]"
    Lamp1 (1054,413 30x30), variable: dIO_ReM.lift[1].roller.err, style: Lamp-Lamp1-Red
    Label (1070,415 132x26), "error"
    Label (891,448 132x26), "roller"
    Line (920,393) (1469,393)
    Line (919,276) (919,906)
    Label (909,635 132x26), "valve_clamp"
    Button (1254,461 130x45), "JOG FW", colour toggle: dIO_ReM.lift[1].roller.forward
        OnMouseDown: execute { dIO_ReM.lift[1].roller.forward := TRUE; }
        OnMouseUp: execute { dIO_ReM.lift[1].roller.forward := FALSE; }
    Button (1253,515 130x45), "JOG BW", colour toggle: dIO_ReM.lift[1].roller.backward
        OnMouseDown: execute { dIO_ReM.lift[1].roller.backward := TRUE; }
        OnMouseUp: execute { dIO_ReM.lift[1].roller.backward := FALSE; }
    Button (1047,475 93x52), "Power On", colour toggle: dIO_ReM.lift[1].roller.Power
        toggle dIO_ReM.lift[1].roller.Power
    Button (1054,590 93x52), "Extend", colour toggle: dIO_ReM.lift[1].valve_clamp.extend
        OnMouseDown: execute { dIO_ReM.lift[1].valve_clamp.extend := TRUE; dIO_ReM.lift[1].valve_clamp.retract := FALSE; }
    Button (1055,666 93x52), "retract", colour toggle: dIO_ReM.lift[1].valve_clamp.retract
        OnMouseDown: execute { dIO_ReM.lift[1].valve_clamp.extend := FALSE; dIO_ReM.lift[1].valve_clamp.retract := TRUE; }
    Lamp1 (1199,603 30x30), variable: dIO_ReM.lift[1].valve_clamp.extended, style: Lamp-Lamp1-Green
    Lamp1 (1201,679 30x30), variable: dIO_ReM.lift[1].valve_clamp.retracted, style: Lamp-Lamp1-Green
    Label (1253,605 132x26), "extended"
    Label (1256,678 132x26), "retracted"
    Line (918,573) (1467,573)
    Line (921,769) (1470,769)
    Label (1506,250 160x26), "valve_perturbation[0]"
    Button (1676,204 93x52), "Extend", colour toggle: dIO_ReM.lift[1].valve_perturbation[0].extend
        OnMouseDown: execute { dIO_ReM.lift[1].valve_perturbation[0].extend := TRUE; dIO_ReM.lift[1].valve_perturbation[0].retract := FALSE; }
    Button (1677,280 93x52), "retract", colour toggle: dIO_ReM.lift[1].valve_perturbation[0].retract
        OnMouseDown: execute { dIO_ReM.lift[1].valve_perturbation[0].extend := FALSE; dIO_ReM.lift[1].valve_perturbation[0].retract := TRUE; }
    Lamp1 (1821,217 30x30), variable: dIO_ReM.lift[1].valve_perturbation[0].extended, style: Lamp-Lamp1-Green
    Lamp1 (1823,293 30x30), variable: dIO_ReM.lift[1].valve_perturbation[0].retracted, style: Lamp-Lamp1-Green
    Label (1875,219 132x26), "extended"
    Label (1878,292 132x26), "retracted"
    Label (1507,415 160x26), "valve_perturbation[1]"
    Button (1677,369 93x52), "Extend", colour toggle: dIO_ReM.lift[1].valve_perturbation[1].extend
        OnMouseDown: execute { dIO_ReM.lift[1].valve_perturbation[1].extend := TRUE; dIO_ReM.lift[1].valve_perturbation[1].retract := FALSE; }
    Button (1678,445 93x52), "retract", colour toggle: dIO_ReM.lift[1].valve_perturbation[1].retract
        OnMouseDown: execute { dIO_ReM.lift[1].valve_perturbation[1].extend := FALSE; dIO_ReM.lift[1].valve_perturbation[1].retract := TRUE; }
    Lamp1 (1822,382 30x30), variable: dIO_ReM.lift[1].valve_perturbation[1].extended, style: Lamp-Lamp1-Green
    Lamp1 (1824,458 30x30), variable: dIO_ReM.lift[1].valve_perturbation[1].retracted, style: Lamp-Lamp1-Green
    Label (1876,384 132x26), "extended"
    Label (1879,457 132x26), "retracted"
    Label (1505,580 160x26), "valve_perturbation[2]"
    Button (1675,534 93x52), "Extend", colour toggle: dIO_ReM.lift[1].valve_perturbation[2].extend
        OnMouseDown: execute { dIO_ReM.lift[1].valve_perturbation[2].extend := TRUE; dIO_ReM.lift[1].valve_perturbation[2].retract := FALSE; }
    Button (1676,610 93x52), "retract", colour toggle: dIO_ReM.lift[1].valve_perturbation[2].retract
        OnMouseDown: execute { dIO_ReM.lift[1].valve_perturbation[2].extend := FALSE; dIO_ReM.lift[1].valve_perturbation[2].retract := TRUE; }
    Lamp1 (1820,547 30x30), variable: dIO_ReM.lift[1].valve_perturbation[2].extended, style: Lamp-Lamp1-Green
    Lamp1 (1822,623 30x30), variable: dIO_ReM.lift[1].valve_perturbation[2].retracted, style: Lamp-Lamp1-Green
    Label (1874,549 132x26), "extended"
    Label (1877,622 132x26), "retracted"
    Label (1501,758 160x26), "valve_perturbation[3]"
    Button (1671,712 93x52), "Extend", colour toggle: dIO_ReM.lift[1].valve_perturbation[3].extend
        OnMouseDown: execute { dIO_ReM.lift[1].valve_perturbation[3].extend := TRUE; dIO_ReM.lift[1].valve_perturbation[3].retract := FALSE; }
    Button (1672,788 93x52), "retract", colour toggle: dIO_ReM.lift[1].valve_perturbation[3].retract
        OnMouseDown: execute { dIO_ReM.lift[1].valve_perturbation[3].extend := FALSE; dIO_ReM.lift[1].valve_perturbation[3].retract := TRUE; }
    Lamp1 (1816,725 30x30), variable: dIO_ReM.lift[1].valve_perturbation[3].extended, style: Lamp-Lamp1-Green
    Lamp1 (1818,801 30x30), variable: dIO_ReM.lift[1].valve_perturbation[3].retracted, style: Lamp-Lamp1-Green
    Label (1870,727 132x26), "extended"
    Label (1873,800 132x26), "retracted"
    Line (1469,273) (1469,906)
    Line (1469,345) (2018,345)
    Line (1471,518) (2020,518)
    Line (1470,693) (2019,693)
    Line (1470,860) (2019,860)
    Line (919,274) (1468,274)
    Line (919,906) (1468,906)
    Label (1256,807 132x26), "NC_contactor"
    Label (919,807 132x26), "axis"
    Button (1053,794 93x52), "Power On", colour toggle: dIO_ReM.lift[1].power_axis
        toggle dIO_ReM.lift[1].power_axis
    Lamp1 (1201,805 30x30), variable: dIO_ReM.lift[1].contactor_axis, style: Lamp-Lamp1-Red
END_VISUALIZATION
